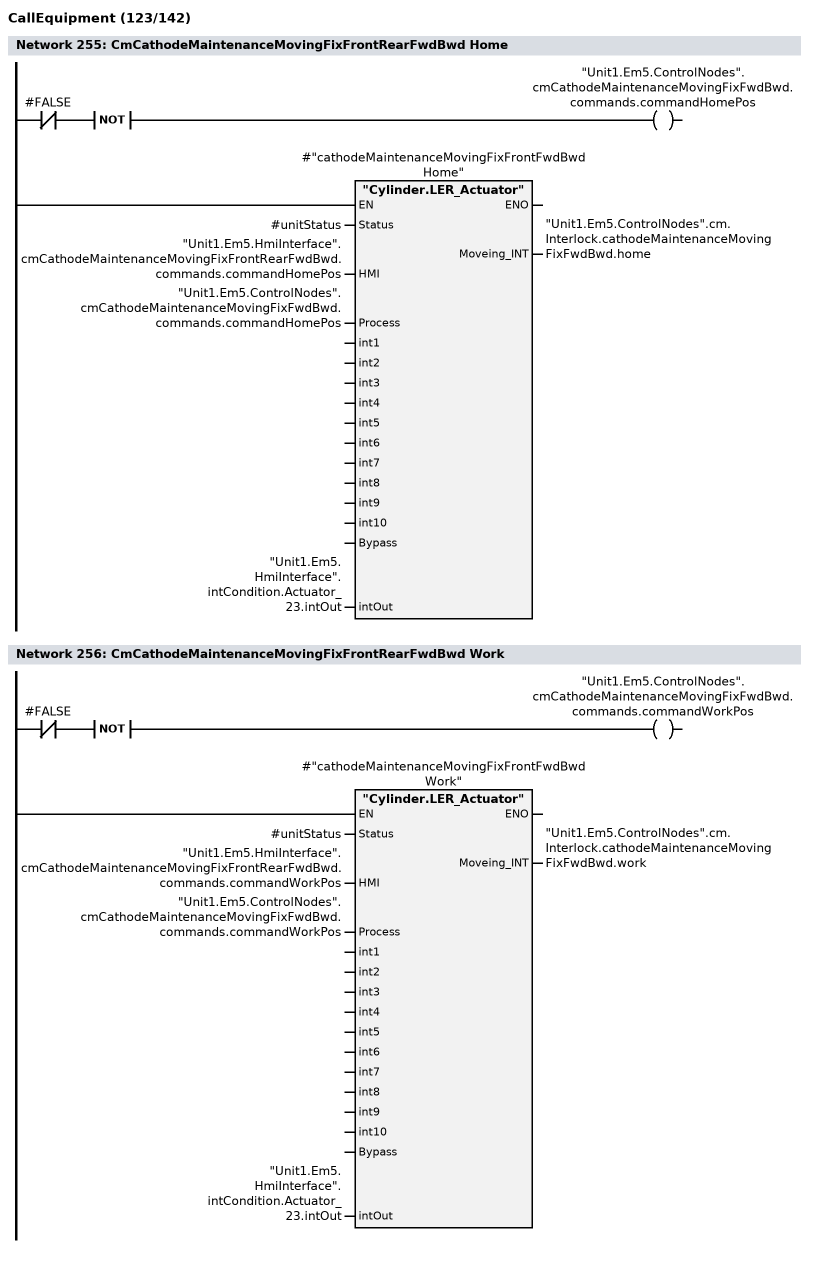
   RUNG wire#powerrail
      I_Contact( #FALSE )
      Not()
      Coil( "Unit1.Em5.ControlNodes".cmCathodeMaintenanceMovingFixFwdBwd.commands.commandHomePos )
   END_RUNG
   RUNG wire#powerrail
      #"cathodeMaintenanceMovingFixFrontFwdBwd Home"(Status := #unitStatus, HMI := "Unit1.Em5.HmiInterface".cmCathodeMaintenanceMovingFixFrontRearFwdBwd.commands.commandHomePos, Process := "Unit1.Em5.ControlNodes".cmCathodeMaintenanceMovingFixFwdBwd.commands.commandHomePos, int1 :=, int2 :=, int3 :=, int4 :=, int5 :=, int6 :=, int7 :=, int8 :=, int9 :=, int10 :=, Bypass :=, intOut := "Unit1.Em5.HmiInterface".intCondition.Actuator_23.intOut, Moveing_INT => "Unit1.Em5.ControlNodes".cm.Interlock.cathodeMaintenanceMovingFixFwdBwd.home)
   END_RUNG
   // the same network as SCL:
   "Unit1.Em5.ControlNodes".cmCathodeMaintenanceMovingFixFwdBwd.commands.commandHomePos := NOT (NOT #FALSE);
   #"cathodeMaintenanceMovingFixFrontFwdBwd Home"(Status := #unitStatus,   // "Cylinder.LER_Actuator"
                           HMI := "Unit1.Em5.HmiInterface".cmCathodeMaintenanceMovingFixFrontRearFwdBwd.commands.commandHomePos,
                           Process := "Unit1.Em5.ControlNodes".cmCathodeMaintenanceMovingFixFwdBwd.commands.commandHomePos,
                           intOut := "Unit1.Em5.HmiInterface".intCondition.Actuator_23.intOut,
                           Moveing_INT => "Unit1.Em5.ControlNodes".cm.Interlock.cathodeMaintenanceMovingFixFwdBwd.home);
END_REGION

REGION Network 256: CmCathodeMaintenanceMovingFixFrontRearFwdBwd Work
   RUNG wire#powerrail
      I_Contact( #FALSE )
      Not()
      Coil( "Unit1.Em5.ControlNodes".cmCathodeMaintenanceMovingFixFwdBwd.commands.commandWorkPos )
   END_RUNG
   RUNG wire#powerrail
      #"cathodeMaintenanceMovingFixFrontFwdBwd Work"(Status := #unitStatus, HMI := "Unit1.Em5.HmiInterface".cmCathodeMaintenanceMovingFixFrontRearFwdBwd.commands.commandWorkPos, Process := "Unit1.Em5.ControlNodes".cmCathodeMaintenanceMovingFixFwdBwd.commands.commandWorkPos, int1 :=, int2 :=, int3 :=, int4 :=, int5 :=, int6 :=, int7 :=, int8 :=, int9 :=, int10 :=, Bypass :=, intOut := "Unit1.Em5.HmiInterface".intCondition.Actuator_23.intOut, Moveing_INT => "Unit1.Em5.ControlNodes".cm.Interlock.cathodeMaintenanceMovingFixFwdBwd.work)
   END_RUNG
   // the same network as SCL:
   "Unit1.Em5.ControlNodes".cmCathodeMaintenanceMovingFixFwdBwd.commands.commandWorkPos := NOT (NOT #FALSE);
   #"cathodeMaintenanceMovingFixFrontFwdBwd Work"(Status := #unitStatus,   // "Cylinder.LER_Actuator"
                           HMI := "Unit1.Em5.HmiInterface".cmCathodeMaintenanceMovingFixFrontRearFwdBwd.commands.commandWorkPos,
                           Process := "Unit1.Em5.ControlNodes".cmCathodeMaintenanceMovingFixFwdBwd.commands.commandWorkPos,
                           intOut := "Unit1.Em5.HmiInterface".intCondition.Actuator_23.intOut,
                           Moveing_INT => "Unit1.Em5.ControlNodes".cm.Interlock.cathodeMaintenanceMovingFixFwdBwd.work);
END_REGION

REGION Network 257: Call instCmCathodeMaintenanceMovingFixFrontRearFwdBwd
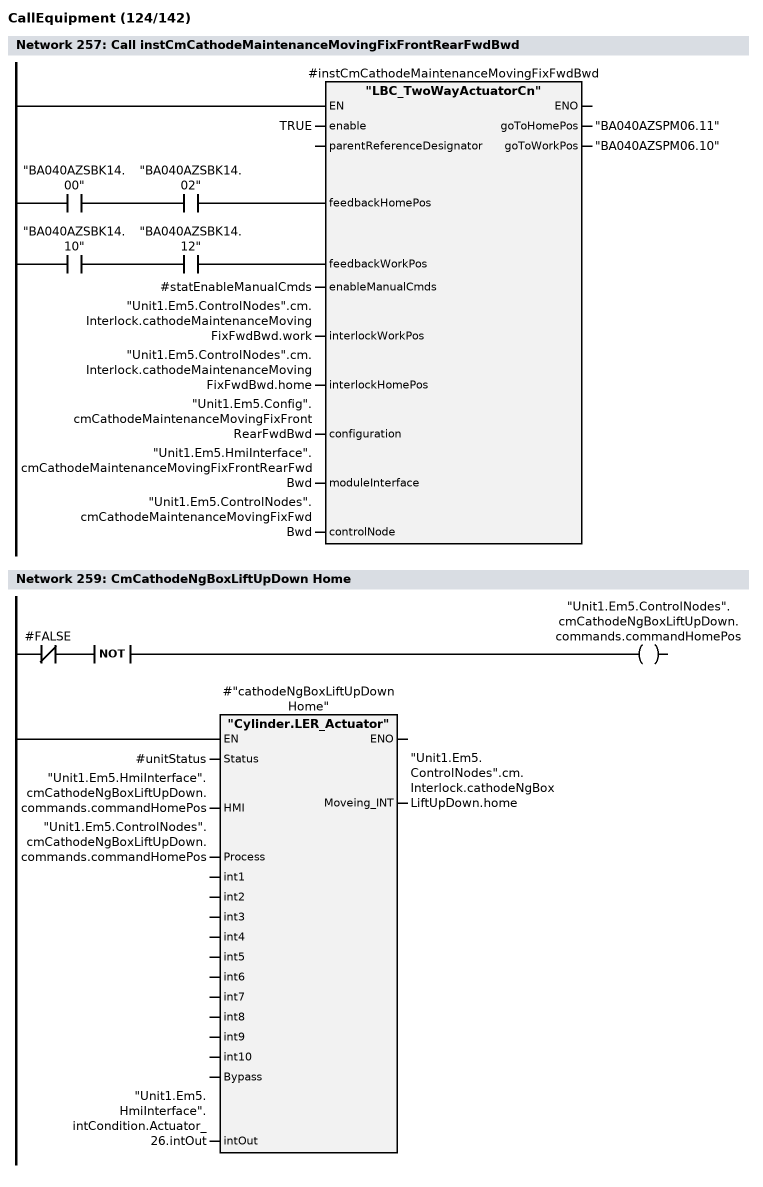
   RUNG wire#powerrail
      #instCmCathodeMaintenanceMovingFixFwdBwd(feedbackHomePos := wire#w1, feedbackWorkPos := wire#w2, enable := TRUE, parentReferenceDesignator :=, enableManualCmds := #statEnableManualCmds, interlockWorkPos := "Unit1.Em5.ControlNodes".cm.Interlock.cathodeMaintenanceMovingFixFwdBwd.work, interlockHomePos := "Unit1.Em5.ControlNodes".cm.Interlock.cathodeMaintenanceMovingFixFwdBwd.home, configuration := "Unit1.Em5.Config".cmCathodeMaintenanceMovingFixFrontRearFwdBwd, moduleInterface := "Unit1.Em5.HmiInterface".cmCathodeMaintenanceMovingFixFrontRearFwdBwd, controlNode := "Unit1.Em5.ControlNodes".cmCathodeMaintenanceMovingFixFwdBwd, goToHomePos => "BA040AZSPM06.11", goToWorkPos => "BA040AZSPM06.10")
   END_RUNG
   RUNG wire#powerrail
      Contact( "BA040AZSBK14.00" )
      Contact( "BA040AZSBK14.02" )
   END_RUNG wire#w1
   RUNG wire#powerrail
      Contact( "BA040AZSBK14.10" )
      Contact( "BA040AZSBK14.12" )
   END_RUNG wire#w2
   // the same network as SCL:
   #instCmCathodeMaintenanceMovingFixFwdBwd(enable := TRUE,   // "LBC_TwoWayActuatorCn"
                           feedbackHomePos := "BA040AZSBK14.00" AND "BA040AZSBK14.02",
                           feedbackWorkPos := "BA040AZSBK14.10" AND "BA040AZSBK14.12",
                           enableManualCmds := #statEnableManualCmds,
                           interlockWorkPos := "Unit1.Em5.ControlNodes".cm.Interlock.cathodeMaintenanceMovingFixFwdBwd.work,
                           interlockHomePos := "Unit1.Em5.ControlNodes".cm.Interlock.cathodeMaintenanceMovingFixFwdBwd.home,
                           configuration := "Unit1.Em5.Config".cmCathodeMaintenanceMovingFixFrontRearFwdBwd,
                           moduleInterface := "Unit1.Em5.HmiInterface".cmCathodeMaintenanceMovingFixFrontRearFwdBwd,
                           controlNode := "Unit1.Em5.ControlNodes".cmCathodeMaintenanceMovingFixFwdBwd,
                           goToHomePos => "BA040AZSPM06.11",
                           goToWorkPos => "BA040AZSPM06.10");
END_REGION

REGION Network 259: CmCathodeNgBoxLiftUpDown Home
   RUNG wire#powerrail
      I_Contact( #FALSE )
      Not()
      Coil( "Unit1.Em5.ControlNodes".cmCathodeNgBoxLiftUpDown.commands.commandHomePos )
   END_RUNG
   RUNG wire#powerrail
      #"cathodeNgBoxLiftUpDown Home"(Status := #unitStatus, HMI := "Unit1.Em5.HmiInterface".cmCathodeNgBoxLiftUpDown.commands.commandHomePos, Process := "Unit1.Em5.ControlNodes".cmCathodeNgBoxLiftUpDown.commands.commandHomePos, int1 :=, int2 :=, int3 :=, int4 :=, int5 :=, int6 :=, int7 :=, int8 :=, int9 :=, int10 :=, Bypass :=, intOut := "Unit1.Em5.HmiInterface".intCondition.Actuator_26.intOut, Moveing_INT => "Unit1.Em5.ControlNodes".cm.Interlock.cathodeNgBoxLiftUpDown.home)
   END_RUNG
   // the same network as SCL:
   "Unit1.Em5.ControlNodes".cmCathodeNgBoxLiftUpDown.commands.commandHomePos := NOT (NOT #FALSE);
   #"cathodeNgBoxLiftUpDown Home"(Status := #unitStatus,   // "Cylinder.LER_Actuator"
                           HMI := "Unit1.Em5.HmiInterface".cmCathodeNgBoxLiftUpDown.commands.commandHomePos,
                           Process := "Unit1.Em5.ControlNodes".cmCathodeNgBoxLiftUpDown.commands.commandHomePos,
                           intOut := "Unit1.Em5.HmiInterface".intCondition.Actuator_26.intOut,
                           Moveing_INT => "Unit1.Em5.ControlNodes".cm.Interlock.cathodeNgBoxLiftUpDown.home);
END_REGION

REGION Network 260: CmCathodeNgBoxLiftUpDown Work
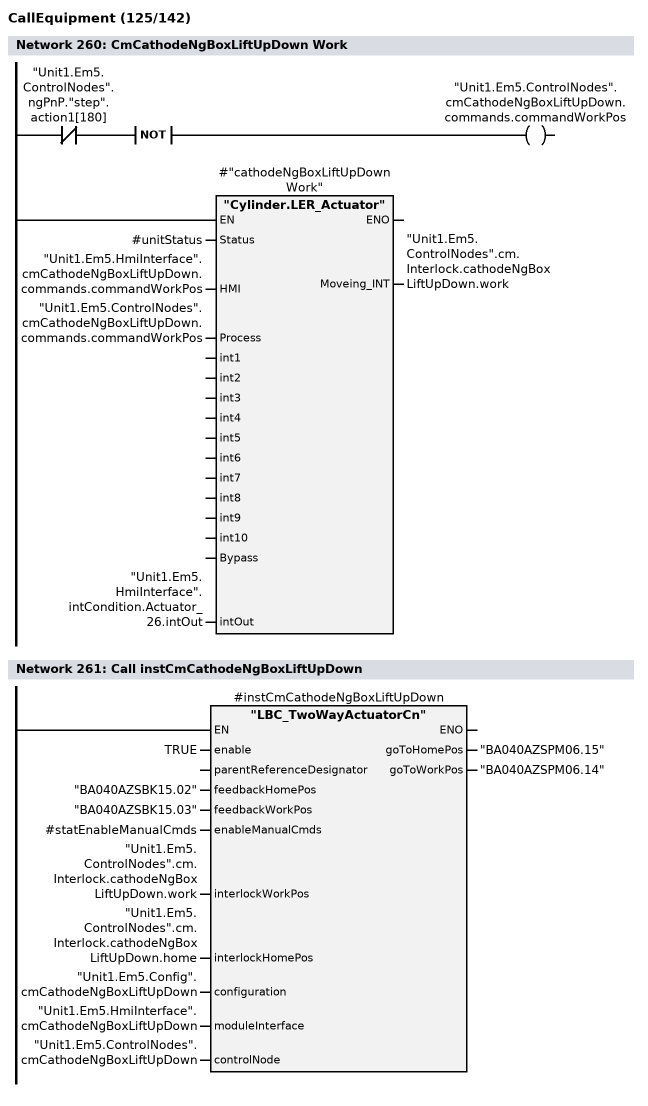
   RUNG wire#powerrail
      I_Contact( "Unit1.Em5.ControlNodes".ngPnP."step".action1[180] )
      Not()
      Coil( "Unit1.Em5.ControlNodes".cmCathodeNgBoxLiftUpDown.commands.commandWorkPos )
   END_RUNG
   RUNG wire#powerrail
      #"cathodeNgBoxLiftUpDown Work"(Status := #unitStatus, HMI := "Unit1.Em5.HmiInterface".cmCathodeNgBoxLiftUpDown.commands.commandWorkPos, Process := "Unit1.Em5.ControlNodes".cmCathodeNgBoxLiftUpDown.commands.commandWorkPos, int1 :=, int2 :=, int3 :=, int4 :=, int5 :=, int6 :=, int7 :=, int8 :=, int9 :=, int10 :=, Bypass :=, intOut := "Unit1.Em5.HmiInterface".intCondition.Actuator_26.intOut, Moveing_INT => "Unit1.Em5.ControlNodes".cm.Interlock.cathodeNgBoxLiftUpDown.work)
   END_RUNG
   // the same network as SCL:
   "Unit1.Em5.ControlNodes".cmCathodeNgBoxLiftUpDown.commands.commandWorkPos := NOT (NOT "Unit1.Em5.ControlNodes".ngPnP."step".action1[180]);
   #"cathodeNgBoxLiftUpDown Work"(Status := #unitStatus,   // "Cylinder.LER_Actuator"
                           HMI := "Unit1.Em5.HmiInterface".cmCathodeNgBoxLiftUpDown.commands.commandWorkPos,
                           Process := "Unit1.Em5.ControlNodes".cmCathodeNgBoxLiftUpDown.commands.commandWorkPos,
                           intOut := "Unit1.Em5.HmiInterface".intCondition.Actuator_26.intOut,
                           Moveing_INT => "Unit1.Em5.ControlNodes".cm.Interlock.cathodeNgBoxLiftUpDown.work);
END_REGION

REGION Network 261: Call instCmCathodeNgBoxLiftUpDown
   RUNG wire#powerrail
      #instCmCathodeNgBoxLiftUpDown(enable := TRUE, parentReferenceDesignator :=, feedbackHomePos := "BA040AZSBK15.02", feedbackWorkPos := "BA040AZSBK15.03", enableManualCmds := #statEnableManualCmds, interlockWorkPos := "Unit1.Em5.ControlNodes".cm.Interlock.cathodeNgBoxLiftUpDown.work, interlockHomePos := "Unit1.Em5.ControlNodes".cm.Interlock.cathodeNgBoxLiftUpDown.home, configuration := "Unit1.Em5.Config".cmCathodeNgBoxLiftUpDown, moduleInterface := "Unit1.Em5.HmiInterface".cmCathodeNgBoxLiftUpDown, controlNode := "Unit1.Em5.ControlNodes".cmCathodeNgBoxLiftUpDown, goToHomePos => "BA040AZSPM06.15", goToWorkPos => "BA040AZSPM06.14")
   END_RUNG
   // the same network as SCL:
   #instCmCathodeNgBoxLiftUpDown(enable := TRUE,   // "LBC_TwoWayActuatorCn"
                           feedbackHomePos := "BA040AZSBK15.02",
                           feedbackWorkPos := "BA040AZSBK15.03",
                           enableManualCmds := #statEnableManualCmds,
                           interlockWorkPos := "Unit1.Em5.ControlNodes".cm.Interlock.cathodeNgBoxLiftUpDown.work,
                           interlockHomePos := "Unit1.Em5.ControlNodes".cm.Interlock.cathodeNgBoxLiftUpDown.home,
                           configuration := "Unit1.Em5.Config".cmCathodeNgBoxLiftUpDown,
                           moduleInterface := "Unit1.Em5.HmiInterface".cmCathodeNgBoxLiftUpDown,
                           controlNode := "Unit1.Em5.ControlNodes".cmCathodeNgBoxLiftUpDown,
                           goToHomePos => "BA040AZSPM06.15",
                           goToWorkPos => "BA040AZSPM06.14");
END_REGION

REGION Network 263: CmCathodeNgBoxLockUpDown Home
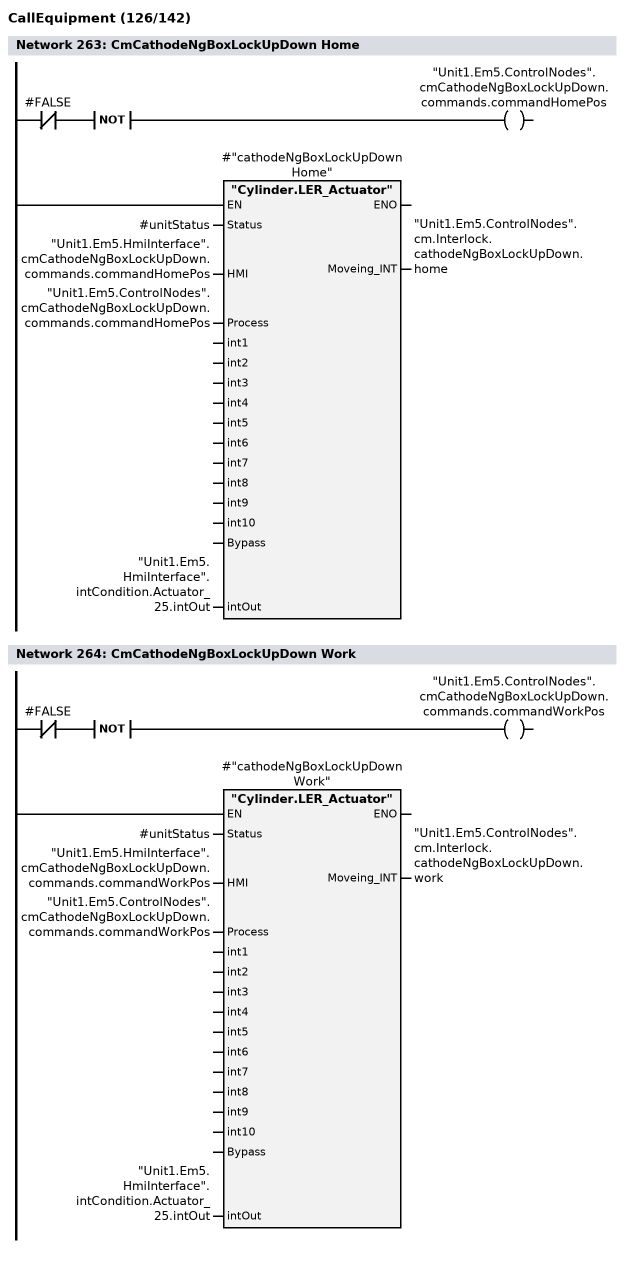
   RUNG wire#powerrail
      I_Contact( #FALSE )
      Not()
      Coil( "Unit1.Em5.ControlNodes".cmCathodeNgBoxLockUpDown.commands.commandHomePos )
   END_RUNG
   RUNG wire#powerrail
      #"cathodeNgBoxLockUpDown Home"(Status := #unitStatus, HMI := "Unit1.Em5.HmiInterface".cmCathodeNgBoxLockUpDown.commands.commandHomePos, Process := "Unit1.Em5.ControlNodes".cmCathodeNgBoxLockUpDown.commands.commandHomePos, int1 :=, int2 :=, int3 :=, int4 :=, int5 :=, int6 :=, int7 :=, int8 :=, int9 :=, int10 :=, Bypass :=, intOut := "Unit1.Em5.HmiInterface".intCondition.Actuator_25.intOut, Moveing_INT => "Unit1.Em5.ControlNodes".cm.Interlock.cathodeNgBoxLockUpDown.home)
   END_RUNG
   // the same network as SCL:
   "Unit1.Em5.ControlNodes".cmCathodeNgBoxLockUpDown.commands.commandHomePos := NOT (NOT #FALSE);
   #"cathodeNgBoxLockUpDown Home"(Status := #unitStatus,   // "Cylinder.LER_Actuator"
                           HMI := "Unit1.Em5.HmiInterface".cmCathodeNgBoxLockUpDown.commands.commandHomePos,
                           Process := "Unit1.Em5.ControlNodes".cmCathodeNgBoxLockUpDown.commands.commandHomePos,
                           intOut := "Unit1.Em5.HmiInterface".intCondition.Actuator_25.intOut,
                           Moveing_INT => "Unit1.Em5.ControlNodes".cm.Interlock.cathodeNgBoxLockUpDown.home);
END_REGION

REGION Network 264: CmCathodeNgBoxLockUpDown Work
   RUNG wire#powerrail
      I_Contact( #FALSE )
      Not()
      Coil( "Unit1.Em5.ControlNodes".cmCathodeNgBoxLockUpDown.commands.commandWorkPos )
   END_RUNG
   RUNG wire#powerrail
      #"cathodeNgBoxLockUpDown Work"(Status := #unitStatus, HMI := "Unit1.Em5.HmiInterface".cmCathodeNgBoxLockUpDown.commands.commandWorkPos, Process := "Unit1.Em5.ControlNodes".cmCathodeNgBoxLockUpDown.commands.commandWorkPos, int1 :=, int2 :=, int3 :=, int4 :=, int5 :=, int6 :=, int7 :=, int8 :=, int9 :=, int10 :=, Bypass :=, intOut := "Unit1.Em5.HmiInterface".intCondition.Actuator_25.intOut, Moveing_INT => "Unit1.Em5.ControlNodes".cm.Interlock.cathodeNgBoxLockUpDown.work)
   END_RUNG
   // the same network as SCL:
   "Unit1.Em5.ControlNodes".cmCathodeNgBoxLockUpDown.commands.commandWorkPos := NOT (NOT #FALSE);
   #"cathodeNgBoxLockUpDown Work"(Status := #unitStatus,   // "Cylinder.LER_Actuator"
                           HMI := "Unit1.Em5.HmiInterface".cmCathodeNgBoxLockUpDown.commands.commandWorkPos,
                           Process := "Unit1.Em5.ControlNodes".cmCathodeNgBoxLockUpDown.commands.commandWorkPos,
                           intOut := "Unit1.Em5.HmiInterface".intCondition.Actuator_25.intOut,
                           Moveing_INT => "Unit1.Em5.ControlNodes".cm.Interlock.cathodeNgBoxLockUpDown.work);
END_REGION

REGION Network 265: Call instCmCathodeNgBoxLockUpDown
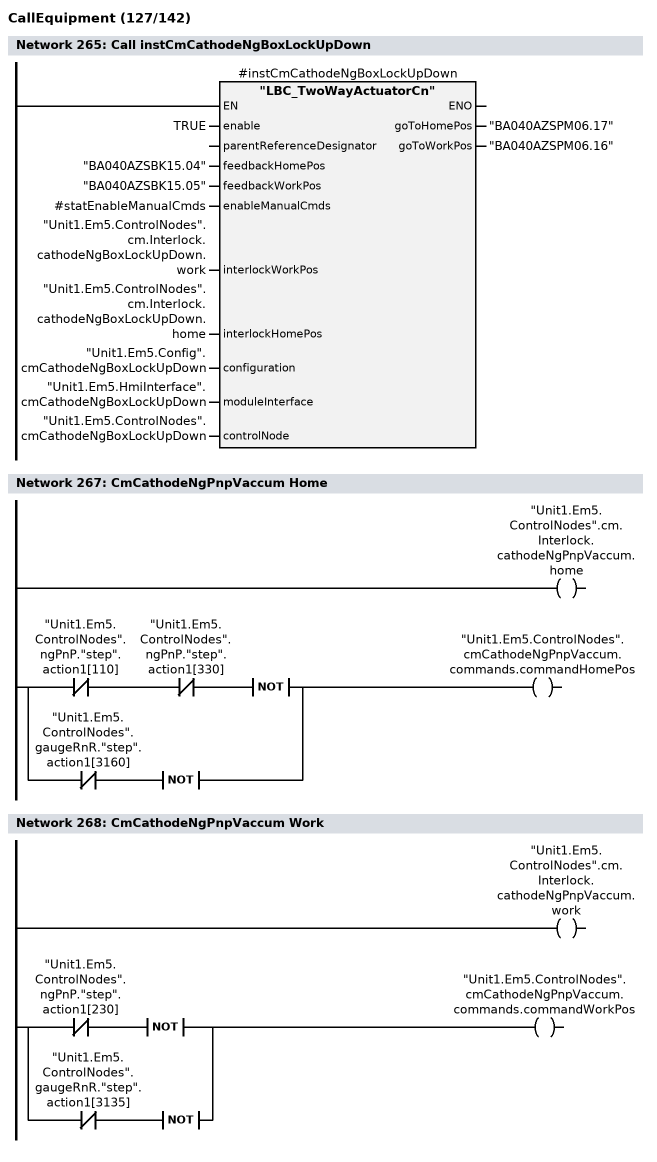
   RUNG wire#powerrail
      #instCmCathodeNgBoxLockUpDown(enable := TRUE, parentReferenceDesignator :=, feedbackHomePos := "BA040AZSBK15.04", feedbackWorkPos := "BA040AZSBK15.05", enableManualCmds := #statEnableManualCmds, interlockWorkPos := "Unit1.Em5.ControlNodes".cm.Interlock.cathodeNgBoxLockUpDown.work, interlockHomePos := "Unit1.Em5.ControlNodes".cm.Interlock.cathodeNgBoxLockUpDown.home, configuration := "Unit1.Em5.Config".cmCathodeNgBoxLockUpDown, moduleInterface := "Unit1.Em5.HmiInterface".cmCathodeNgBoxLockUpDown, controlNode := "Unit1.Em5.ControlNodes".cmCathodeNgBoxLockUpDown, goToHomePos => "BA040AZSPM06.17", goToWorkPos => "BA040AZSPM06.16")
   END_RUNG
   // the same network as SCL:
   #instCmCathodeNgBoxLockUpDown(enable := TRUE,   // "LBC_TwoWayActuatorCn"
                           feedbackHomePos := "BA040AZSBK15.04",
                           feedbackWorkPos := "BA040AZSBK15.05",
                           enableManualCmds := #statEnableManualCmds,
                           interlockWorkPos := "Unit1.Em5.ControlNodes".cm.Interlock.cathodeNgBoxLockUpDown.work,
                           interlockHomePos := "Unit1.Em5.ControlNodes".cm.Interlock.cathodeNgBoxLockUpDown.home,
                           configuration := "Unit1.Em5.Config".cmCathodeNgBoxLockUpDown,
                           moduleInterface := "Unit1.Em5.HmiInterface".cmCathodeNgBoxLockUpDown,
                           controlNode := "Unit1.Em5.ControlNodes".cmCathodeNgBoxLockUpDown,
                           goToHomePos => "BA040AZSPM06.17",
                           goToWorkPos => "BA040AZSPM06.16");
END_REGION

REGION Network 267: CmCathodeNgPnpVaccum Home
   RUNG wire#powerrail
      Coil( "Unit1.Em5.ControlNodes".cm.Interlock.cathodeNgPnpVaccum.home )
   END_RUNG
   RUNG wire#powerrail
      I_Contact( "Unit1.Em5.ControlNodes".ngPnP."step".action1[110] )
      I_Contact( "Unit1.Em5.ControlNodes".ngPnP."step".action1[330] )
      Not()
      wire#w1
      Coil( "Unit1.Em5.ControlNodes".cmCathodeNgPnpVaccum.commands.commandHomePos )
   END_RUNG
   RUNG wire#powerrail
      I_Contact( "Unit1.Em5.ControlNodes".gaugeRnR."step".action1[3160] )
      Not()
   END_RUNG wire#w1
   // the same network as SCL:
   "Unit1.Em5.ControlNodes".cm.Interlock.cathodeNgPnpVaccum.home := TRUE;
   "Unit1.Em5.ControlNodes".cmCathodeNgPnpVaccum.commands.commandHomePos := NOT (NOT "Unit1.Em5.ControlNodes".ngPnP."step".action1[110] AND NOT "Unit1.Em5.ControlNodes".ngPnP."step".action1[330]) OR NOT (NOT "Unit1.Em5.ControlNodes".gaugeRnR."step".action1[3160]);
END_REGION

REGION Network 268: CmCathodeNgPnpVaccum Work
   RUNG wire#powerrail
      Coil( "Unit1.Em5.ControlNodes".cm.Interlock.cathodeNgPnpVaccum.work )
   END_RUNG
   RUNG wire#powerrail
      I_Contact( "Unit1.Em5.ControlNodes".ngPnP."step".action1[230] )
      Not()
      wire#w1
      Coil( "Unit1.Em5.ControlNodes".cmCathodeNgPnpVaccum.commands.commandWorkPos )
   END_RUNG
   RUNG wire#powerrail
      I_Contact( "Unit1.Em5.ControlNodes".gaugeRnR."step".action1[3135] )
      Not()
   END_RUNG wire#w1
   // the same network as SCL:
   "Unit1.Em5.ControlNodes".cm.Interlock.cathodeNgPnpVaccum.work := TRUE;
   "Unit1.Em5.ControlNodes".cmCathodeNgPnpVaccum.commands.commandWorkPos := NOT (NOT "Unit1.Em5.ControlNodes".ngPnP."step".action1[230]) OR NOT (NOT "Unit1.Em5.ControlNodes".gaugeRnR."step".action1[3135]);
END_REGION

REGION Network 269: Call instCmCathodeNgPnpVaccum
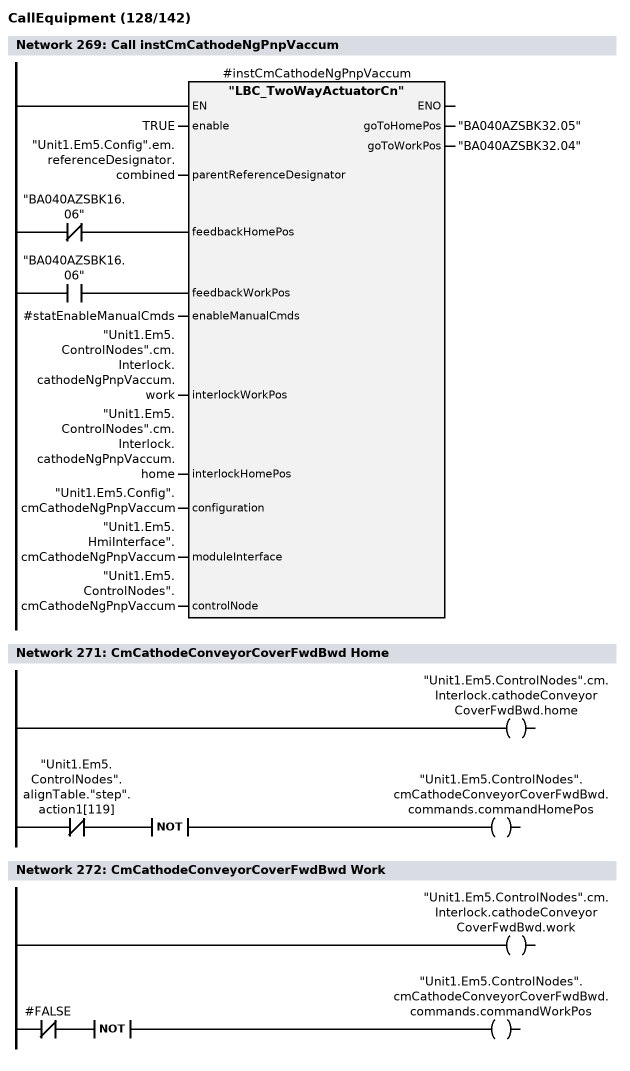
   RUNG wire#powerrail
      #instCmCathodeNgPnpVaccum(feedbackHomePos := wire#w1, feedbackWorkPos := wire#w2, enable := TRUE, parentReferenceDesignator := "Unit1.Em5.Config".em.referenceDesignator.combined, enableManualCmds := #statEnableManualCmds, interlockWorkPos := "Unit1.Em5.ControlNodes".cm.Interlock.cathodeNgPnpVaccum.work, interlockHomePos := "Unit1.Em5.ControlNodes".cm.Interlock.cathodeNgPnpVaccum.home, configuration := "Unit1.Em5.Config".cmCathodeNgPnpVaccum, moduleInterface := "Unit1.Em5.HmiInterface".cmCathodeNgPnpVaccum, controlNode := "Unit1.Em5.ControlNodes".cmCathodeNgPnpVaccum, goToHomePos => "BA040AZSBK32.05", goToWorkPos => "BA040AZSBK32.04")
   END_RUNG
   RUNG wire#powerrail
      I_Contact( "BA040AZSBK16.06" )
   END_RUNG wire#w1
   RUNG wire#powerrail
      Contact( "BA040AZSBK16.06" )
   END_RUNG wire#w2
   // the same network as SCL:
   #instCmCathodeNgPnpVaccum(enable := TRUE,   // "LBC_TwoWayActuatorCn"
                           parentReferenceDesignator := "Unit1.Em5.Config".em.referenceDesignator.combined,
                           feedbackHomePos := NOT "BA040AZSBK16.06",
                           feedbackWorkPos := "BA040AZSBK16.06",
                           enableManualCmds := #statEnableManualCmds,
                           interlockWorkPos := "Unit1.Em5.ControlNodes".cm.Interlock.cathodeNgPnpVaccum.work,
                           interlockHomePos := "Unit1.Em5.ControlNodes".cm.Interlock.cathodeNgPnpVaccum.home,
                           configuration := "Unit1.Em5.Config".cmCathodeNgPnpVaccum,
                           moduleInterface := "Unit1.Em5.HmiInterface".cmCathodeNgPnpVaccum,
                           controlNode := "Unit1.Em5.ControlNodes".cmCathodeNgPnpVaccum,
                           goToHomePos => "BA040AZSBK32.05",
                           goToWorkPos => "BA040AZSBK32.04");
END_REGION

REGION Network 271: CmCathodeConveyorCoverFwdBwd Home
   RUNG wire#powerrail
      Coil( "Unit1.Em5.ControlNodes".cm.Interlock.cathodeConveyorCoverFwdBwd.home )
   END_RUNG
   RUNG wire#powerrail
      I_Contact( "Unit1.Em5.ControlNodes".alignTable."step".action1[119] )
      Not()
      Coil( "Unit1.Em5.ControlNodes".cmCathodeConveyorCoverFwdBwd.commands.commandHomePos )
   END_RUNG
   // the same network as SCL:
   "Unit1.Em5.ControlNodes".cm.Interlock.cathodeConveyorCoverFwdBwd.home := TRUE;
   "Unit1.Em5.ControlNodes".cmCathodeConveyorCoverFwdBwd.commands.commandHomePos := NOT (NOT "Unit1.Em5.ControlNodes".alignTable."step".action1[119]);
END_REGION

REGION Network 272: CmCathodeConveyorCoverFwdBwd Work
   RUNG wire#powerrail
      Coil( "Unit1.Em5.ControlNodes".cm.Interlock.cathodeConveyorCoverFwdBwd.work )
   END_RUNG
   RUNG wire#powerrail
      I_Contact( #FALSE )
      Not()
      Coil( "Unit1.Em5.ControlNodes".cmCathodeConveyorCoverFwdBwd.commands.commandWorkPos )
   END_RUNG
   // the same network as SCL:
   "Unit1.Em5.ControlNodes".cm.Interlock.cathodeConveyorCoverFwdBwd.work := TRUE;
   "Unit1.Em5.ControlNodes".cmCathodeConveyorCoverFwdBwd.commands.commandWorkPos := NOT (NOT #FALSE);
END_REGION

REGION Network 273: Call instCmCathodeConveyorCoverFwdBwd
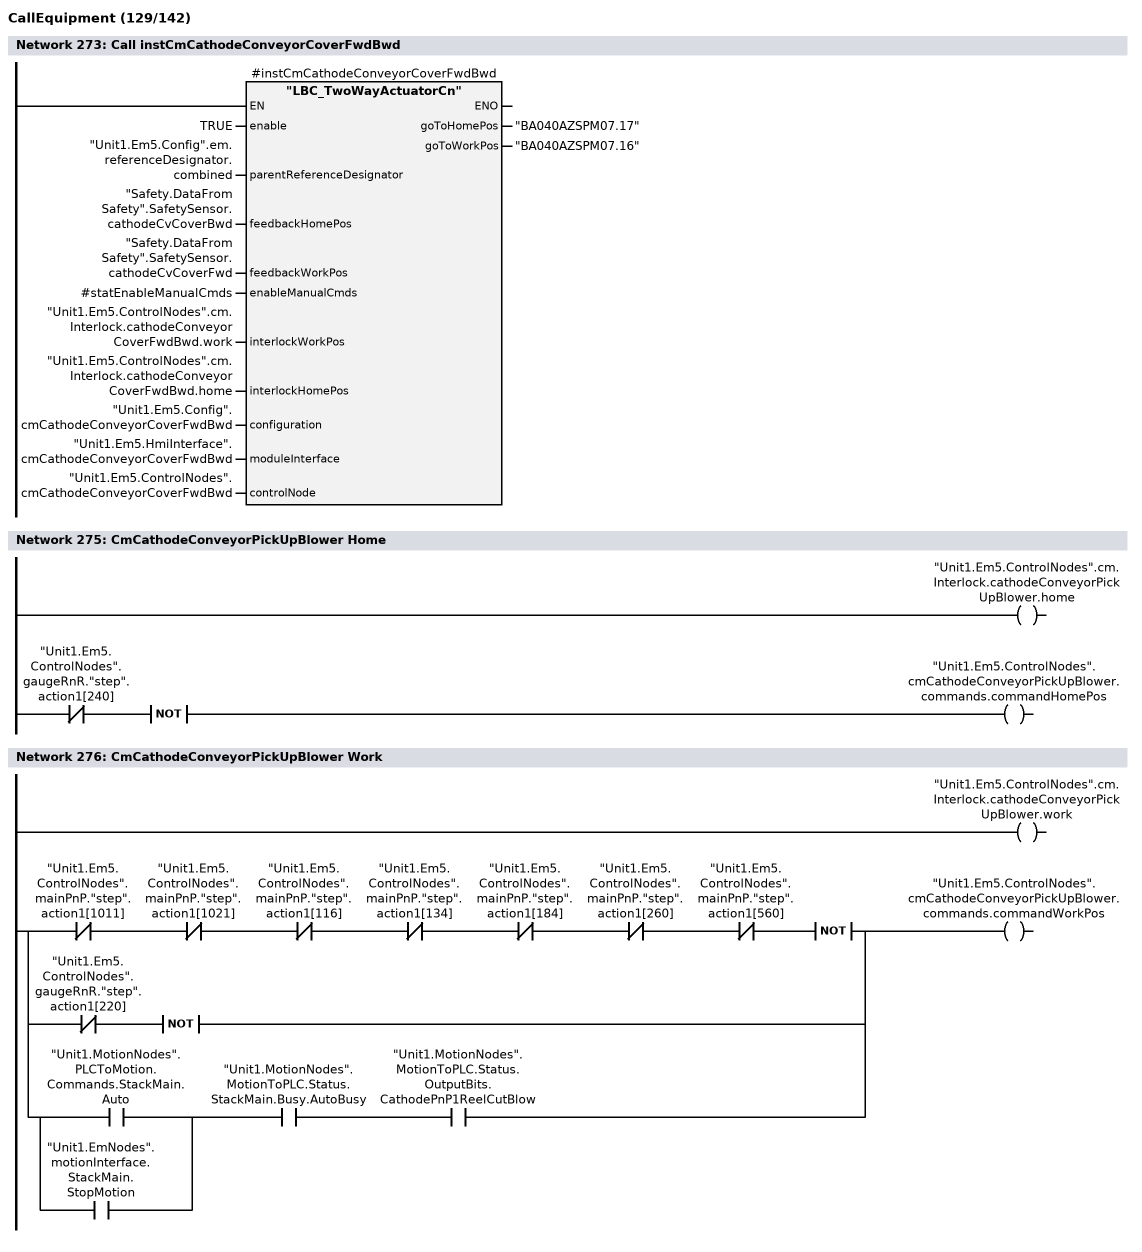
   RUNG wire#powerrail
      #instCmCathodeConveyorCoverFwdBwd(enable := TRUE, parentReferenceDesignator := "Unit1.Em5.Config".em.referenceDesignator.combined, feedbackHomePos := "Safety.DataFromSafety".SafetySensor.cathodeCvCoverBwd, feedbackWorkPos := "Safety.DataFromSafety".SafetySensor.cathodeCvCoverFwd, enableManualCmds := #statEnableManualCmds, interlockWorkPos := "Unit1.Em5.ControlNodes".cm.Interlock.cathodeConveyorCoverFwdBwd.work, interlockHomePos := "Unit1.Em5.ControlNodes".cm.Interlock.cathodeConveyorCoverFwdBwd.home, configuration := "Unit1.Em5.Config".cmCathodeConveyorCoverFwdBwd, moduleInterface := "Unit1.Em5.HmiInterface".cmCathodeConveyorCoverFwdBwd, controlNode := "Unit1.Em5.ControlNodes".cmCathodeConveyorCoverFwdBwd, goToHomePos => "BA040AZSPM07.17", goToWorkPos => "BA040AZSPM07.16")
   END_RUNG
   // the same network as SCL:
   #instCmCathodeConveyorCoverFwdBwd(enable := TRUE,   // "LBC_TwoWayActuatorCn"
                           parentReferenceDesignator := "Unit1.Em5.Config".em.referenceDesignator.combined,
                           feedbackHomePos := "Safety.DataFromSafety".SafetySensor.cathodeCvCoverBwd,
                           feedbackWorkPos := "Safety.DataFromSafety".SafetySensor.cathodeCvCoverFwd,
                           enableManualCmds := #statEnableManualCmds,
                           interlockWorkPos := "Unit1.Em5.ControlNodes".cm.Interlock.cathodeConveyorCoverFwdBwd.work,
                           interlockHomePos := "Unit1.Em5.ControlNodes".cm.Interlock.cathodeConveyorCoverFwdBwd.home,
                           configuration := "Unit1.Em5.Config".cmCathodeConveyorCoverFwdBwd,
                           moduleInterface := "Unit1.Em5.HmiInterface".cmCathodeConveyorCoverFwdBwd,
                           controlNode := "Unit1.Em5.ControlNodes".cmCathodeConveyorCoverFwdBwd,
                           goToHomePos => "BA040AZSPM07.17",
                           goToWorkPos => "BA040AZSPM07.16");
END_REGION

REGION Network 275: CmCathodeConveyorPickUpBlower Home
   RUNG wire#powerrail
      Coil( "Unit1.Em5.ControlNodes".cm.Interlock.cathodeConveyorPickUpBlower.home )
   END_RUNG
   RUNG wire#powerrail
      I_Contact( "Unit1.Em5.ControlNodes".gaugeRnR."step".action1[240] )
      Not()
      Coil( "Unit1.Em5.ControlNodes".cmCathodeConveyorPickUpBlower.commands.commandHomePos )
   END_RUNG
   // the same network as SCL:
   "Unit1.Em5.ControlNodes".cm.Interlock.cathodeConveyorPickUpBlower.home := TRUE;
   "Unit1.Em5.ControlNodes".cmCathodeConveyorPickUpBlower.commands.commandHomePos := NOT (NOT "Unit1.Em5.ControlNodes".gaugeRnR."step".action1[240]);
END_REGION

REGION Network 276: CmCathodeConveyorPickUpBlower Work
   RUNG wire#powerrail
      Coil( "Unit1.Em5.ControlNodes".cm.Interlock.cathodeConveyorPickUpBlower.work )
   END_RUNG
   RUNG wire#powerrail
      I_Contact( "Unit1.Em5.ControlNodes".mainPnP."step".action1[1011] )
      I_Contact( "Unit1.Em5.ControlNodes".mainPnP."step".action1[1021] )
      I_Contact( "Unit1.Em5.ControlNodes".mainPnP."step".action1[116] )
      I_Contact( "Unit1.Em5.ControlNodes".mainPnP."step".action1[134] )
      I_Contact( "Unit1.Em5.ControlNodes".mainPnP."step".action1[184] )
      I_Contact( "Unit1.Em5.ControlNodes".mainPnP."step".action1[260] )
      I_Contact( "Unit1.Em5.ControlNodes".mainPnP."step".action1[560] )
      Not()
      wire#w1
      Coil( "Unit1.Em5.ControlNodes".cmCathodeConveyorPickUpBlower.commands.commandWorkPos )
   END_RUNG
   RUNG wire#powerrail
      I_Contact( "Unit1.Em5.ControlNodes".gaugeRnR."step".action1[220] )
      Not()
   END_RUNG wire#w1
   RUNG wire#powerrail
      Contact( "Unit1.MotionNodes".PLCToMotion.Commands.StackMain.Auto )
      wire#w2
      Contact( "Unit1.MotionNodes".MotionToPLC.Status.StackMain.Busy.AutoBusy )
      Contact( "Unit1.MotionNodes".MotionToPLC.Status.OutputBits.CathodePnP1ReelCutBlow )
   END_RUNG wire#w1
   RUNG wire#powerrail
      Contact( "Unit1.EmNodes".motionInterface.StackMain.StopMotion )
   END_RUNG wire#w2
   // the same network as SCL:
   "Unit1.Em5.ControlNodes".cm.Interlock.cathodeConveyorPickUpBlower.work := TRUE;
   "Unit1.Em5.ControlNodes".cmCathodeConveyorPickUpBlower.commands.commandWorkPos := NOT (NOT "Unit1.Em5.ControlNodes".mainPnP."step".action1[1011] AND NOT "Unit1.Em5.ControlNodes".mainPnP."step".action1[1021] AND NOT "Unit1.Em5.ControlNodes".mainPnP."step".action1[116] AND NOT "Unit1.Em5.ControlNodes".mainPnP."step".action1[134] AND NOT "Unit1.Em5.ControlNodes".mainPnP."step".action1[184] AND NOT "Unit1.Em5.ControlNodes".mainPnP."step".action1[260] AND NOT "Unit1.Em5.ControlNodes".mainPnP."step".action1[560]) OR NOT (NOT "Unit1.Em5.ControlNodes".gaugeRnR."step".action1[220]) OR (("Unit1.MotionNodes".PLCToMotion.Commands.StackMain.Auto OR "Unit1.EmNodes".motionInterface.StackMain.StopMotion) AND "Unit1.MotionNodes".MotionToPLC.Status.StackMain.Busy.AutoBusy AND "Unit1.MotionNodes".MotionToPLC.Status.OutputBits.CathodePnP1ReelCutBlow);
END_REGION

REGION Network 277: Call instCmCathodeConveyorPickUpBlower
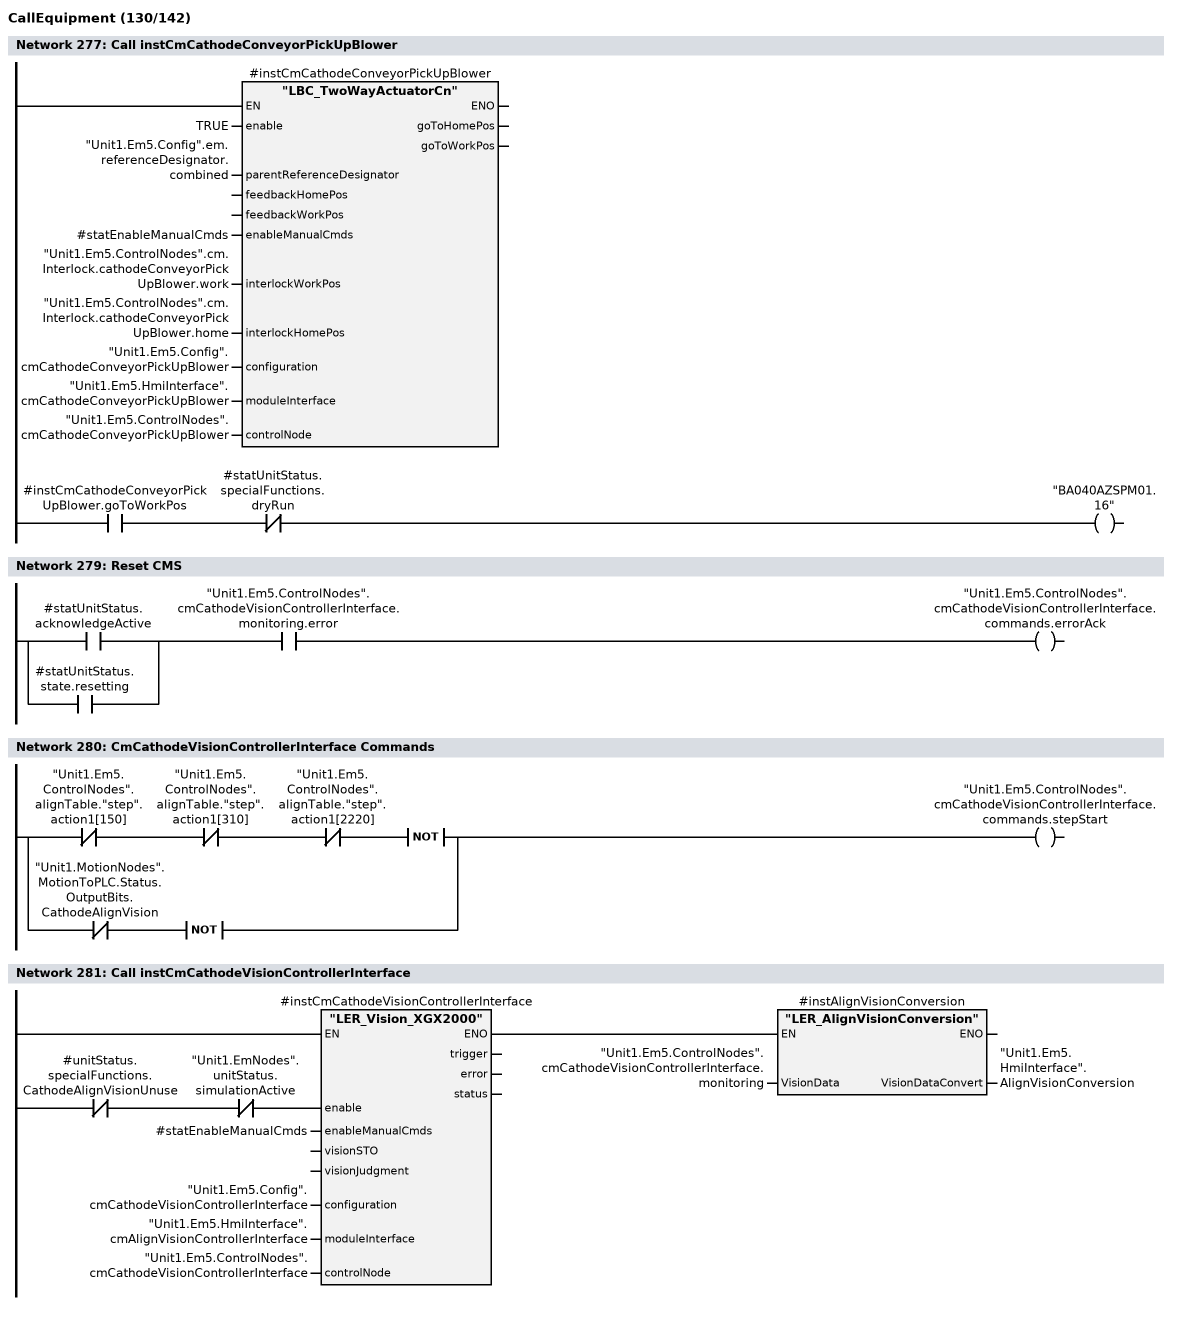
   RUNG wire#powerrail
      #instCmCathodeConveyorPickUpBlower(enable := TRUE, parentReferenceDesignator := "Unit1.Em5.Config".em.referenceDesignator.combined, feedbackHomePos :=, feedbackWorkPos :=, enableManualCmds := #statEnableManualCmds, interlockWorkPos := "Unit1.Em5.ControlNodes".cm.Interlock.cathodeConveyorPickUpBlower.work, interlockHomePos := "Unit1.Em5.ControlNodes".cm.Interlock.cathodeConveyorPickUpBlower.home, configuration := "Unit1.Em5.Config".cmCathodeConveyorPickUpBlower, moduleInterface := "Unit1.Em5.HmiInterface".cmCathodeConveyorPickUpBlower, controlNode := "Unit1.Em5.ControlNodes".cmCathodeConveyorPickUpBlower, goToHomePos =>, goToWorkPos =>)
   END_RUNG
   RUNG wire#powerrail
      Contact( #instCmCathodeConveyorPickUpBlower.goToWorkPos )
      I_Contact( #statUnitStatus.specialFunctions.dryRun )
      Coil( "BA040AZSPM01.16" )
   END_RUNG
   // the same network as SCL:
   #instCmCathodeConveyorPickUpBlower(enable := TRUE,   // "LBC_TwoWayActuatorCn"
                           parentReferenceDesignator := "Unit1.Em5.Config".em.referenceDesignator.combined,
                           enableManualCmds := #statEnableManualCmds,
                           interlockWorkPos := "Unit1.Em5.ControlNodes".cm.Interlock.cathodeConveyorPickUpBlower.work,
                           interlockHomePos := "Unit1.Em5.ControlNodes".cm.Interlock.cathodeConveyorPickUpBlower.home,
                           configuration := "Unit1.Em5.Config".cmCathodeConveyorPickUpBlower,
                           moduleInterface := "Unit1.Em5.HmiInterface".cmCathodeConveyorPickUpBlower,
                           controlNode := "Unit1.Em5.ControlNodes".cmCathodeConveyorPickUpBlower);
   "BA040AZSPM01.16" := #instCmCathodeConveyorPickUpBlower.goToWorkPos AND NOT #statUnitStatus.specialFunctions.dryRun;
END_REGION

REGION Network 278: ******************** Control Modules (Accessories) ********************
END_REGION

REGION Network 279: Reset CMS
   RUNG wire#powerrail
      Contact( #statUnitStatus.acknowledgeActive )
      wire#w1
      Contact( "Unit1.Em5.ControlNodes".cmCathodeVisionControllerInterface.monitoring.error )
      Coil( "Unit1.Em5.ControlNodes".cmCathodeVisionControllerInterface.commands.errorAck )
   END_RUNG
   RUNG wire#powerrail
      Contact( #statUnitStatus.state.resetting )
   END_RUNG wire#w1
   // the same network as SCL:
   "Unit1.Em5.ControlNodes".cmCathodeVisionControllerInterface.commands.errorAck := (#statUnitStatus.acknowledgeActive OR #statUnitStatus.state.resetting) AND "Unit1.Em5.ControlNodes".cmCathodeVisionControllerInterface.monitoring.error;
END_REGION

REGION Network 280: CmCathodeVisionControllerInterface Commands
   RUNG wire#powerrail
      I_Contact( "Unit1.Em5.ControlNodes".alignTable."step".action1[150] )
      I_Contact( "Unit1.Em5.ControlNodes".alignTable."step".action1[310] )
      I_Contact( "Unit1.Em5.ControlNodes".alignTable."step".action1[2220] )
      Not()
      wire#w1
      Coil( "Unit1.Em5.ControlNodes".cmCathodeVisionControllerInterface.commands.stepStart )
   END_RUNG
   RUNG wire#powerrail
      I_Contact( "Unit1.MotionNodes".MotionToPLC.Status.OutputBits.CathodeAlignVision )
      Not()
   END_RUNG wire#w1
   // the same network as SCL:
   "Unit1.Em5.ControlNodes".cmCathodeVisionControllerInterface.commands.stepStart := NOT (NOT "Unit1.Em5.ControlNodes".alignTable."step".action1[150] AND NOT "Unit1.Em5.ControlNodes".alignTable."step".action1[310] AND NOT "Unit1.Em5.ControlNodes".alignTable."step".action1[2220]) OR NOT (NOT "Unit1.MotionNodes".MotionToPLC.Status.OutputBits.CathodeAlignVision);
END_REGION

REGION Network 281: Call instCmCathodeVisionControllerInterface
   RUNG wire#powerrail
      #instCmCathodeVisionControllerInterface(enable := wire#w1, enableManualCmds := #statEnableManualCmds, visionSTO :=, visionJudgment :=, configuration := "Unit1.Em5.Config".cmCathodeVisionControllerInterface, moduleInterface := "Unit1.Em5.HmiInterface".cmAlignVisionControllerInterface, controlNode := "Unit1.Em5.ControlNodes".cmCathodeVisionControllerInterface, trigger =>, error =>, status =>)
      #instAlignVisionConversion(VisionData := "Unit1.Em5.ControlNodes".cmCathodeVisionControllerInterface.monitoring, VisionDataConvert => "Unit1.Em5.HmiInterface".AlignVisionConversion)
   END_RUNG
   RUNG wire#powerrail
      I_Contact( #unitStatus.specialFunctions.CathodeAlignVisionUnuse )
      I_Contact( "Unit1.EmNodes".unitStatus.simulationActive )
   END_RUNG wire#w1
   // the same network as SCL:
   #instCmCathodeVisionControllerInterface(enable := NOT #unitStatus.specialFunctions.CathodeAlignVisionUnuse AND NOT "Unit1.EmNodes".unitStatus.simulationActive,   // "LER_Vision_XGX2000"
                           enableManualCmds := #statEnableManualCmds,
                           configuration := "Unit1.Em5.Config".cmCathodeVisionControllerInterface,
                           moduleInterface := "Unit1.Em5.HmiInterface".cmAlignVisionControllerInterface,
                           controlNode := "Unit1.Em5.ControlNodes".cmCathodeVisionControllerInterface,
                           ENO => #_w1);
   IF #_w1 THEN
       #instAlignVisionConversion(VisionData := "Unit1.Em5.ControlNodes".cmCathodeVisionControllerInterface.monitoring,   // "LER_AlignVisionConversion"
                               VisionDataConvert => "Unit1.Em5.HmiInterface".AlignVisionConversion);
   END_IF;
END_REGION

REGION Network 282: *************** Feedback to Unit ***************************
END_REGION

REGION Network 283: Determine StateComplete (SC) in Mode Production
   // Conditions for the Equipment Modules "stateComplete" feedback to the unit. This feedback is given when the task in for the respective state is complete.
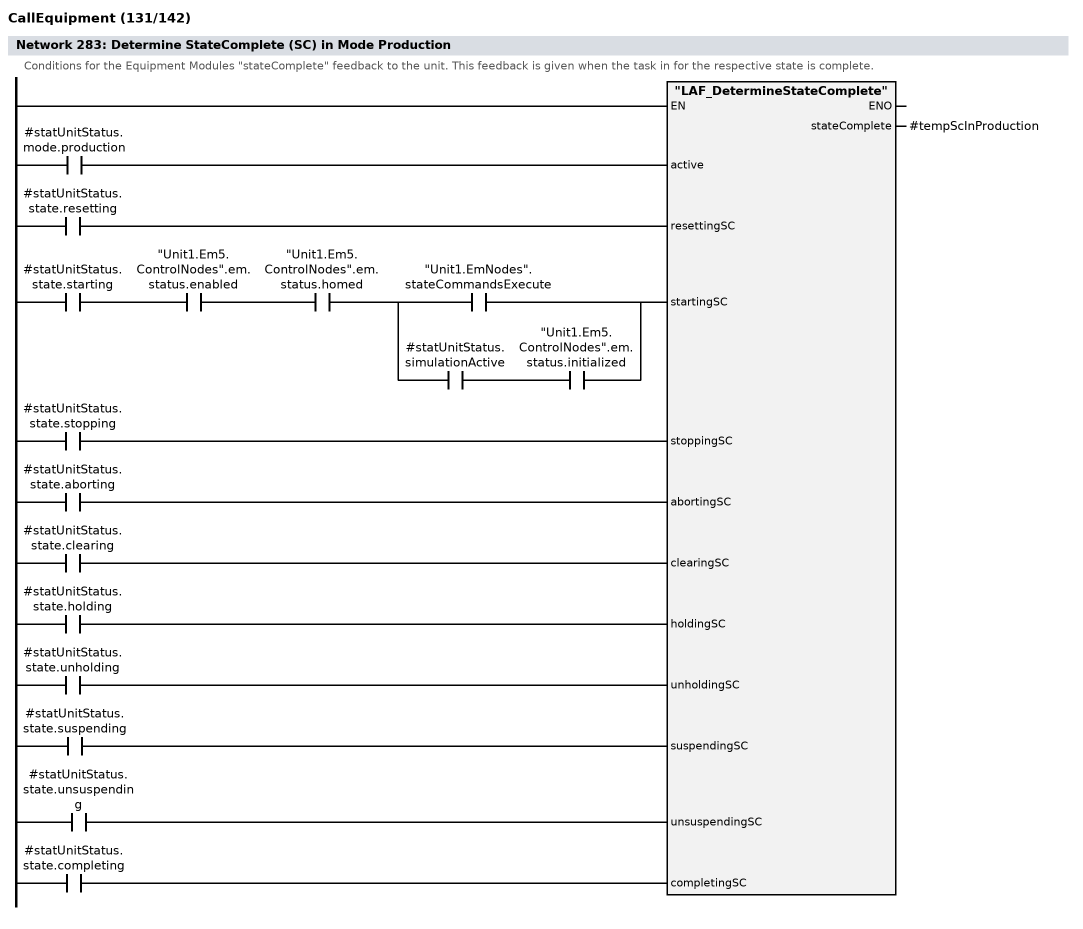
   RUNG wire#powerrail
      "LAF_DetermineStateComplete"(active := wire#w1, resettingSC := wire#w2, startingSC := wire#w4, stoppingSC := wire#w5, abortingSC := wire#w6, clearingSC := wire#w7, holdingSC := wire#w8, unholdingSC := wire#w9, suspendingSC := wire#w10, unsuspendingSC := wire#w11, completingSC := wire#w12, stateComplete => #tempScInProduction)
   END_RUNG
   RUNG wire#powerrail
      Contact( #statUnitStatus.mode.production )
   END_RUNG wire#w1
   RUNG wire#powerrail
      Contact( #statUnitStatus.state.resetting )
   END_RUNG wire#w2
   RUNG wire#powerrail
      Contact( #statUnitStatus.state.starting )
      Contact( "Unit1.Em5.ControlNodes".em.status.enabled )
      Contact( "Unit1.Em5.ControlNodes".em.status.homed )
      wire#w3
      Contact( "Unit1.EmNodes".stateCommandsExecute )
   END_RUNG wire#w4
   RUNG wire#w3
      Contact( #statUnitStatus.simulationActive )
      Contact( "Unit1.Em5.ControlNodes".em.status.initialized )
   END_RUNG wire#w4
   RUNG wire#powerrail
      Contact( #statUnitStatus.state.stopping )
   END_RUNG wire#w5
   RUNG wire#powerrail
      Contact( #statUnitStatus.state.aborting )
   END_RUNG wire#w6
   RUNG wire#powerrail
      Contact( #statUnitStatus.state.clearing )
   END_RUNG wire#w7
   RUNG wire#powerrail
      Contact( #statUnitStatus.state.holding )
   END_RUNG wire#w8
   RUNG wire#powerrail
      Contact( #statUnitStatus.state.unholding )
   END_RUNG wire#w9
   RUNG wire#powerrail
      Contact( #statUnitStatus.state.suspending )
   END_RUNG wire#w10
   RUNG wire#powerrail
      Contact( #statUnitStatus.state.unsuspending )
   END_RUNG wire#w11
   RUNG wire#powerrail
      Contact( #statUnitStatus.state.completing )
   END_RUNG wire#w12
   // the same network as SCL:
   "LAF_DetermineStateComplete"(active := #statUnitStatus.mode.production,
                           resettingSC := #statUnitStatus.state.resetting,
                           startingSC := #statUnitStatus.state.starting AND "Unit1.Em5.ControlNodes".em.status.enabled AND "Unit1.Em5.ControlNodes".em.status.homed AND ("Unit1.EmNodes".stateCommandsExecute OR (#statUnitStatus.simulationActive AND "Unit1.Em5.ControlNodes".em.status.initialized)),
                           stoppingSC := #statUnitStatus.state.stopping,
                           abortingSC := #statUnitStatus.state.aborting,
                           clearingSC := #statUnitStatus.state.clearing,
                           holdingSC := #statUnitStatus.state.holding,
                           unholdingSC := #statUnitStatus.state.unholding,
                           suspendingSC := #statUnitStatus.state.suspending,
                           unsuspendingSC := #statUnitStatus.state.unsuspending,
                           completingSC := #statUnitStatus.state.completing,
                           stateComplete => #tempScInProduction);
END_REGION

REGION Network 284: Determine StateComplete (SC) in Mode Maintenance/Manual
   // Conditions for the Equipment Modules "stateComplete" feedback to the unit. This feedback is given when the task in for the respective state is complete.
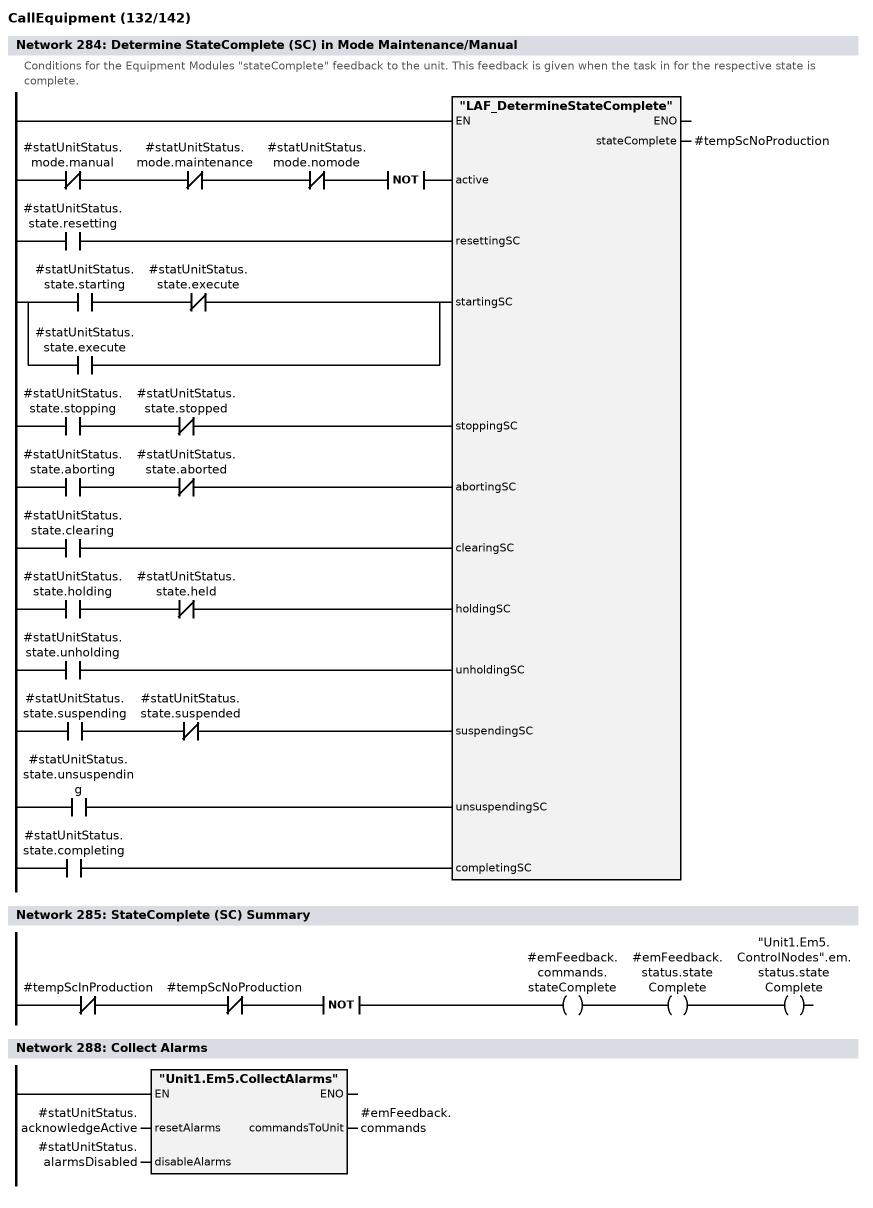
   RUNG wire#powerrail
      "LAF_DetermineStateComplete"(active := wire#w1, resettingSC := wire#w2, startingSC := wire#w3, stoppingSC := wire#w4, abortingSC := wire#w5, clearingSC := wire#w6, holdingSC := wire#w7, unholdingSC := wire#w8, suspendingSC := wire#w9, unsuspendingSC := wire#w10, completingSC := wire#w11, stateComplete => #tempScNoProduction)
   END_RUNG
   RUNG wire#powerrail
      I_Contact( #statUnitStatus.mode.manual )
      I_Contact( #statUnitStatus.mode.maintenance )
      I_Contact( #statUnitStatus.mode.nomode )
      Not()
   END_RUNG wire#w1
   RUNG wire#powerrail
      Contact( #statUnitStatus.state.resetting )
   END_RUNG wire#w2
   RUNG wire#powerrail
      Contact( #statUnitStatus.state.starting )
      I_Contact( #statUnitStatus.state.execute )
   END_RUNG wire#w3
   RUNG wire#powerrail
      Contact( #statUnitStatus.state.execute )
   END_RUNG wire#w3
   RUNG wire#powerrail
      Contact( #statUnitStatus.state.stopping )
      I_Contact( #statUnitStatus.state.stopped )
   END_RUNG wire#w4
   RUNG wire#powerrail
      Contact( #statUnitStatus.state.aborting )
      I_Contact( #statUnitStatus.state.aborted )
   END_RUNG wire#w5
   RUNG wire#powerrail
      Contact( #statUnitStatus.state.clearing )
   END_RUNG wire#w6
   RUNG wire#powerrail
      Contact( #statUnitStatus.state.holding )
      I_Contact( #statUnitStatus.state.held )
   END_RUNG wire#w7
   RUNG wire#powerrail
      Contact( #statUnitStatus.state.unholding )
   END_RUNG wire#w8
   RUNG wire#powerrail
      Contact( #statUnitStatus.state.suspending )
      I_Contact( #statUnitStatus.state.suspended )
   END_RUNG wire#w9
   RUNG wire#powerrail
      Contact( #statUnitStatus.state.unsuspending )
   END_RUNG wire#w10
   RUNG wire#powerrail
      Contact( #statUnitStatus.state.completing )
   END_RUNG wire#w11
   // the same network as SCL:
   "LAF_DetermineStateComplete"(active := NOT (NOT #statUnitStatus.mode.manual AND NOT #statUnitStatus.mode.maintenance AND NOT #statUnitStatus.mode.nomode),
                           resettingSC := #statUnitStatus.state.resetting,
                           startingSC := (#statUnitStatus.state.starting AND NOT #statUnitStatus.state.execute) OR #statUnitStatus.state.execute,
                           stoppingSC := #statUnitStatus.state.stopping AND NOT #statUnitStatus.state.stopped,
                           abortingSC := #statUnitStatus.state.aborting AND NOT #statUnitStatus.state.aborted,
                           clearingSC := #statUnitStatus.state.clearing,
                           holdingSC := #statUnitStatus.state.holding AND NOT #statUnitStatus.state.held,
                           unholdingSC := #statUnitStatus.state.unholding,
                           suspendingSC := #statUnitStatus.state.suspending AND NOT #statUnitStatus.state.suspended,
                           unsuspendingSC := #statUnitStatus.state.unsuspending,
                           completingSC := #statUnitStatus.state.completing,
                           stateComplete => #tempScNoProduction);
END_REGION

REGION Network 285: StateComplete (SC) Summary
   RUNG wire#powerrail
      I_Contact( #tempScInProduction )
      I_Contact( #tempScNoProduction )
      Not()
      Coil( #emFeedback.commands.stateComplete )
      Coil( #emFeedback.status.stateComplete )
      Coil( "Unit1.Em5.ControlNodes".em.status.stateComplete )
   END_RUNG
   // the same network as SCL:
   #emFeedback.commands.stateComplete := NOT (NOT #tempScInProduction AND NOT #tempScNoProduction);
   #emFeedback.status.stateComplete := #emFeedback.commands.stateComplete;
   "Unit1.Em5.ControlNodes".em.status.stateComplete := #emFeedback.commands.stateComplete;
END_REGION

REGION Network 287: *************** Alarms **********************************
END_REGION

REGION Network 288: Collect Alarms
   RUNG wire#powerrail
      "Unit1.Em5.CollectAlarms"(resetAlarms := #statUnitStatus.acknowledgeActive, disableAlarms := #statUnitStatus.alarmsDisabled, commandsToUnit => #emFeedback.commands)
   END_RUNG
   // the same network as SCL:
   "Unit1.Em5.CollectAlarms"(resetAlarms := #statUnitStatus.acknowledgeActive,
                           disableAlarms := #statUnitStatus.alarmsDisabled,
                           commandsToUnit => #emFeedback.commands);
END_REGION

REGION Network 289: Manage Alarms
   // Derive commands from the ProDiag supervision. The ProDiag supervisions contain categories which define the reaction of these supervisions (e.g. abort, stop, hold). These are handed over as commands to the unit level.
   // Alternatively, if no ProDiag should be used, you can use the LAF_ManageBitAlarms to realize bit alarm handling. This block can be found in LAF in folder 70_AlarmHandling.
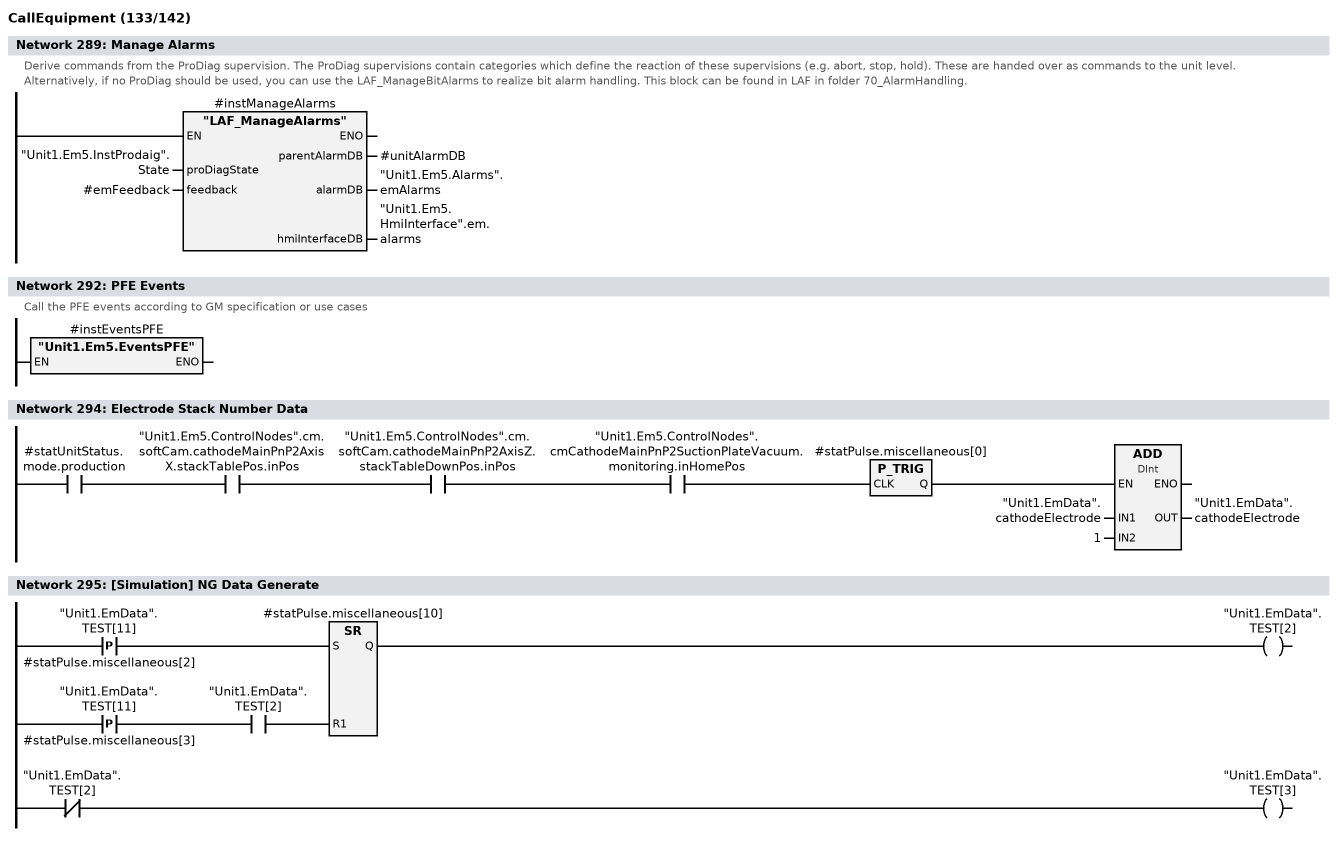
   RUNG wire#powerrail
      #instManageAlarms(proDiagState := "Unit1.Em5.InstProdaig".State, feedback := #emFeedback, parentAlarmDB => #unitAlarmDB, alarmDB => "Unit1.Em5.Alarms".emAlarms, hmiInterfaceDB => "Unit1.Em5.HmiInterface".em.alarms)
   END_RUNG
   // the same network as SCL:
   #instManageAlarms(proDiagState := "Unit1.Em5.InstProdaig".State,   // "LAF_ManageAlarms"
                     feedback := #emFeedback,
                     parentAlarmDB => #unitAlarmDB,
                     alarmDB => "Unit1.Em5.Alarms".emAlarms,
                     hmiInterfaceDB => "Unit1.Em5.HmiInterface".em.alarms);
END_REGION

REGION Network 291: *************** PFE Events**********************************
END_REGION

REGION Network 292: PFE Events
   // Call the PFE events according to GM specification or use cases
   RUNG wire#powerrail
      #instEventsPFE()
   END_RUNG
   // the same network as SCL:
   #instEventsPFE();   // "Unit1.Em5.EventsPFE"
END_REGION

REGION Network 293: ******************** Part Data ********************
END_REGION

REGION Network 294: Electrode Stack Number Data
   RUNG wire#powerrail
      Contact( #statUnitStatus.mode.production )
      Contact( "Unit1.Em5.ControlNodes".cm.softCam.cathodeMainPnP2AxisX.stackTablePos.inPos )
      Contact( "Unit1.Em5.ControlNodes".cm.softCam.cathodeMainPnP2AxisZ.stackTableDownPos.inPos )
      Contact( "Unit1.Em5.ControlNodes".cmCathodeMainPnP2SuctionPlateVacuum.monitoring.inHomePos )
      P_Trig( #statPulse.miscellaneous[0] )
      { S7_Templates := "SrcType := DInt" } Add(in1 := "Unit1.EmData".cathodeElectrode, in2 := 1, out => "Unit1.EmData".cathodeElectrode)
   END_RUNG
   // the same network as SCL:
   #_w1 := #statUnitStatus.mode.production AND "Unit1.Em5.ControlNodes".cm.softCam.cathodeMainPnP2AxisX.stackTablePos.inPos AND "Unit1.Em5.ControlNodes".cm.softCam.cathodeMainPnP2AxisZ.stackTableDownPos.inPos AND "Unit1.Em5.ControlNodes".cmCathodeMainPnP2SuctionPlateVacuum.monitoring.inHomePos;
   #_w2 := #_w1 AND NOT #statPulse.miscellaneous[0];   // rising edge
   #statPulse.miscellaneous[0] := #_w1;
   IF #_w2 THEN "Unit1.EmData".cathodeElectrode := "Unit1.EmData".cathodeElectrode + 1; END_IF;
END_REGION

REGION Network 295: [Simulation] NG Data Generate
   RUNG wire#powerrail
      P_Contact(operand := "Unit1.EmData".TEST[11], bit := #statPulse.miscellaneous[2])
      S_SR(operand := #statPulse.miscellaneous[10], r1 := wire#w1)
      Coil( "Unit1.EmData".TEST[2] )
   END_RUNG
   RUNG wire#powerrail
      P_Contact(operand := "Unit1.EmData".TEST[11], bit := #statPulse.miscellaneous[3])
      Contact( "Unit1.EmData".TEST[2] )
   END_RUNG wire#w1
   RUNG wire#powerrail
      I_Contact( "Unit1.EmData".TEST[2] )
      Coil( "Unit1.EmData".TEST[3] )
   END_RUNG
   // the same network as SCL:
   #_w1 := "Unit1.EmData".TEST[11] AND NOT #statPulse.miscellaneous[2];   // rising edge of "Unit1.EmData".TEST[11]
   #statPulse.miscellaneous[2] := "Unit1.EmData".TEST[11];
   #_w2 := "Unit1.EmData".TEST[11] AND NOT #statPulse.miscellaneous[3];   // rising edge of "Unit1.EmData".TEST[11]
   #statPulse.miscellaneous[3] := "Unit1.EmData".TEST[11];
   IF #_w1 THEN
       #statPulse.miscellaneous[10] := TRUE;   // SR flip-flop
   END_IF;
   IF #_w2 AND "Unit1.EmData".TEST[2] THEN #statPulse.miscellaneous[10] := FALSE; END_IF;
   "Unit1.EmData".TEST[2] := #statPulse.miscellaneous[10];
   "Unit1.EmData".TEST[3] := NOT "Unit1.EmData".TEST[2];
END_REGION

REGION Network 296: Align Vision Data
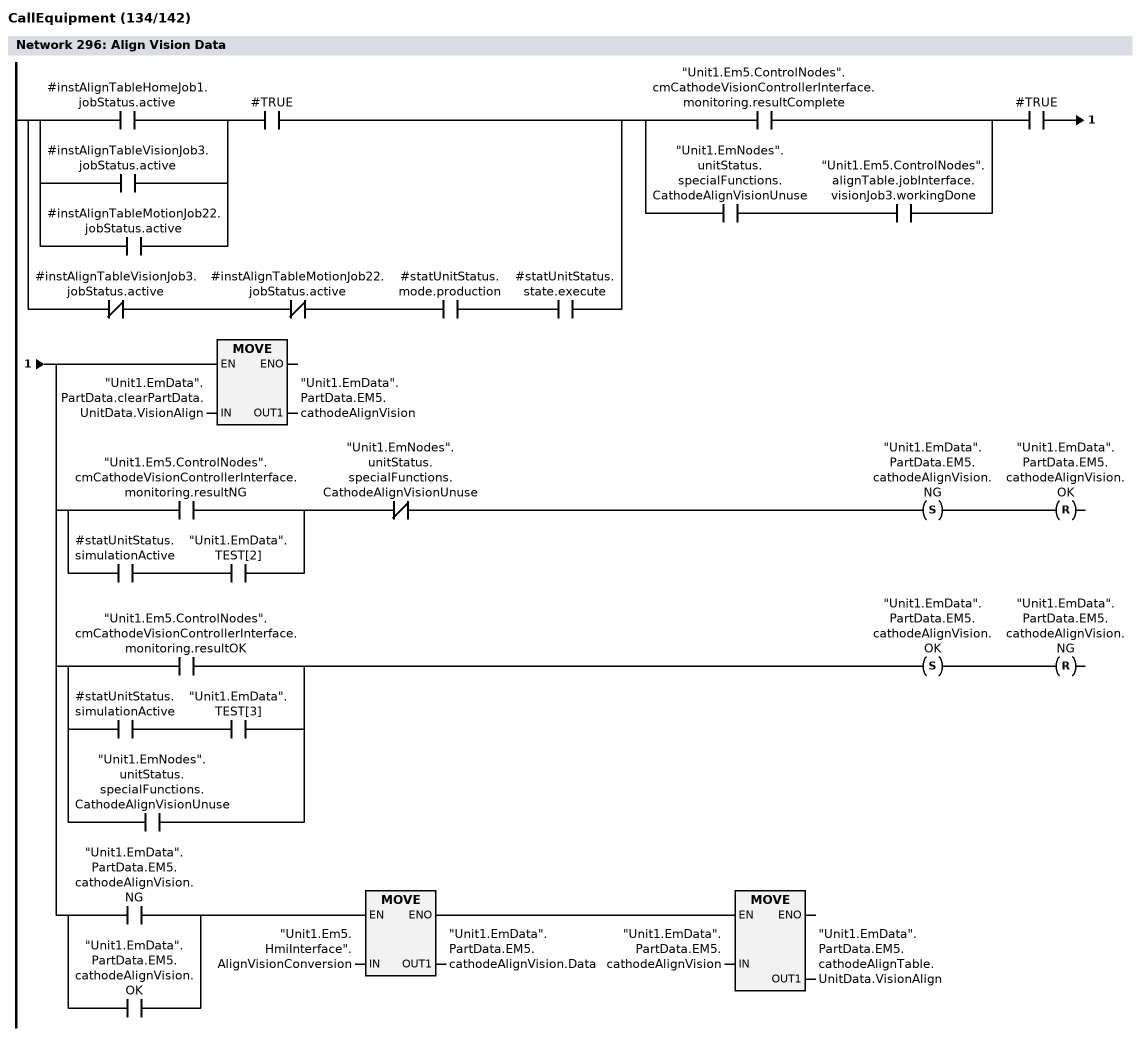
   RUNG wire#powerrail
      Contact( #instAlignTableHomeJob1.jobStatus.active )
      wire#w1
      Contact( #TRUE )
      wire#w2
      Contact( "Unit1.Em5.ControlNodes".cmCathodeVisionControllerInterface.monitoring.resultComplete )
      wire#w3
      Contact( #TRUE )
      wire#w4
      Move(in := "Unit1.EmData".PartData.clearPartData.UnitData.VisionAlign, out1 => "Unit1.EmData".PartData.EM5.cathodeAlignVision)
   END_RUNG
   RUNG wire#powerrail
      Contact( #instAlignTableVisionJob3.jobStatus.active )
   END_RUNG wire#w1
   RUNG wire#powerrail
      Contact( #instAlignTableMotionJob22.jobStatus.active )
   END_RUNG wire#w1
   RUNG wire#powerrail
      I_Contact( #instAlignTableVisionJob3.jobStatus.active )
      I_Contact( #instAlignTableMotionJob22.jobStatus.active )
      Contact( #statUnitStatus.mode.production )
      Contact( #statUnitStatus.state.execute )
   END_RUNG wire#w2
   RUNG wire#w2
      Contact( "Unit1.EmNodes".unitStatus.specialFunctions.CathodeAlignVisionUnuse )
      Contact( "Unit1.Em5.ControlNodes".alignTable.jobInterface.visionJob3.workingDone )
   END_RUNG wire#w3
   RUNG wire#w4
      Contact( "Unit1.Em5.ControlNodes".cmCathodeVisionControllerInterface.monitoring.resultNG )
      wire#w5
      I_Contact( "Unit1.EmNodes".unitStatus.specialFunctions.CathodeAlignVisionUnuse )
      S_Coil( "Unit1.EmData".PartData.EM5.cathodeAlignVision.NG )
      R_Coil( "Unit1.EmData".PartData.EM5.cathodeAlignVision.OK )
   END_RUNG
   RUNG wire#w4
      Contact( #statUnitStatus.simulationActive )
      Contact( "Unit1.EmData".TEST[2] )
   END_RUNG wire#w5
   RUNG wire#w4
      Contact( "Unit1.Em5.ControlNodes".cmCathodeVisionControllerInterface.monitoring.resultOK )
      wire#w6
      S_Coil( "Unit1.EmData".PartData.EM5.cathodeAlignVision.OK )
      R_Coil( "Unit1.EmData".PartData.EM5.cathodeAlignVision.NG )
   END_RUNG
   RUNG wire#w4
      Contact( #statUnitStatus.simulationActive )
      Contact( "Unit1.EmData".TEST[3] )
   END_RUNG wire#w6
   RUNG wire#w4
      Contact( "Unit1.EmNodes".unitStatus.specialFunctions.CathodeAlignVisionUnuse )
   END_RUNG wire#w6
   RUNG wire#w4
      Contact( "Unit1.EmData".PartData.EM5.cathodeAlignVision.NG )
      wire#w7
      Move(in := "Unit1.Em5.HmiInterface".AlignVisionConversion, out1 => "Unit1.EmData".PartData.EM5.cathodeAlignVision.Data)
      Move(in := "Unit1.EmData".PartData.EM5.cathodeAlignVision, out1 => "Unit1.EmData".PartData.EM5.cathodeAlignTable.UnitData.VisionAlign)
   END_RUNG
   RUNG wire#w4
      Contact( "Unit1.EmData".PartData.EM5.cathodeAlignVision.OK )
   END_RUNG wire#w7
   // the same network as SCL:
   #_w1 := (((#instAlignTableHomeJob1.jobStatus.active OR #instAlignTableVisionJob3.jobStatus.active OR #instAlignTableMotionJob22.jobStatus.active) AND #TRUE) OR (NOT #instAlignTableVisionJob3.jobStatus.active AND NOT #instAlignTableMotionJob22.jobStatus.active AND #statUnitStatus.mode.production AND #statUnitStatus.state.execute)) AND ("Unit1.Em5.ControlNodes".cmCathodeVisionControllerInterface.monitoring.resultComplete OR ("Unit1.EmNodes".unitStatus.specialFunctions.CathodeAlignVisionUnuse AND "Unit1.Em5.ControlNodes".alignTable.jobInterface.visionJob3.workingDone)) AND #TRUE;
   IF #_w1 THEN
       "Unit1.EmData".PartData.EM5.cathodeAlignVision := "Unit1.EmData".PartData.clearPartData.UnitData.VisionAlign;
   END_IF;
   IF #_w1 AND ("Unit1.Em5.ControlNodes".cmCathodeVisionControllerInterface.monitoring.resultNG OR (#statUnitStatus.simulationActive AND "Unit1.EmData".TEST[2])) AND NOT "Unit1.EmNodes".unitStatus.specialFunctions.CathodeAlignVisionUnuse THEN
       "Unit1.EmData".PartData.EM5.cathodeAlignVision.NG := TRUE;
       "Unit1.EmData".PartData.EM5.cathodeAlignVision.OK := FALSE;
   END_IF;
   IF #_w1 AND ("Unit1.Em5.ControlNodes".cmCathodeVisionControllerInterface.monitoring.resultOK OR (#statUnitStatus.simulationActive AND "Unit1.EmData".TEST[3]) OR "Unit1.EmNodes".unitStatus.specialFunctions.CathodeAlignVisionUnuse) THEN
       "Unit1.EmData".PartData.EM5.cathodeAlignVision.OK := TRUE;
       "Unit1.EmData".PartData.EM5.cathodeAlignVision.NG := FALSE;
   END_IF;
   IF #_w1 AND ("Unit1.EmData".PartData.EM5.cathodeAlignVision.NG OR "Unit1.EmData".PartData.EM5.cathodeAlignVision.OK) THEN
       "Unit1.EmData".PartData.EM5.cathodeAlignVision.Data := "Unit1.Em5.HmiInterface".AlignVisionConversion;
       "Unit1.EmData".PartData.EM5.cathodeAlignTable.UnitData.VisionAlign := "Unit1.EmData".PartData.EM5.cathodeAlignVision;
   END_IF;
END_REGION

REGION Network 297: ******************** Unit Output ********************
END_REGION

REGION Network 298: Em Nodes Brake Test
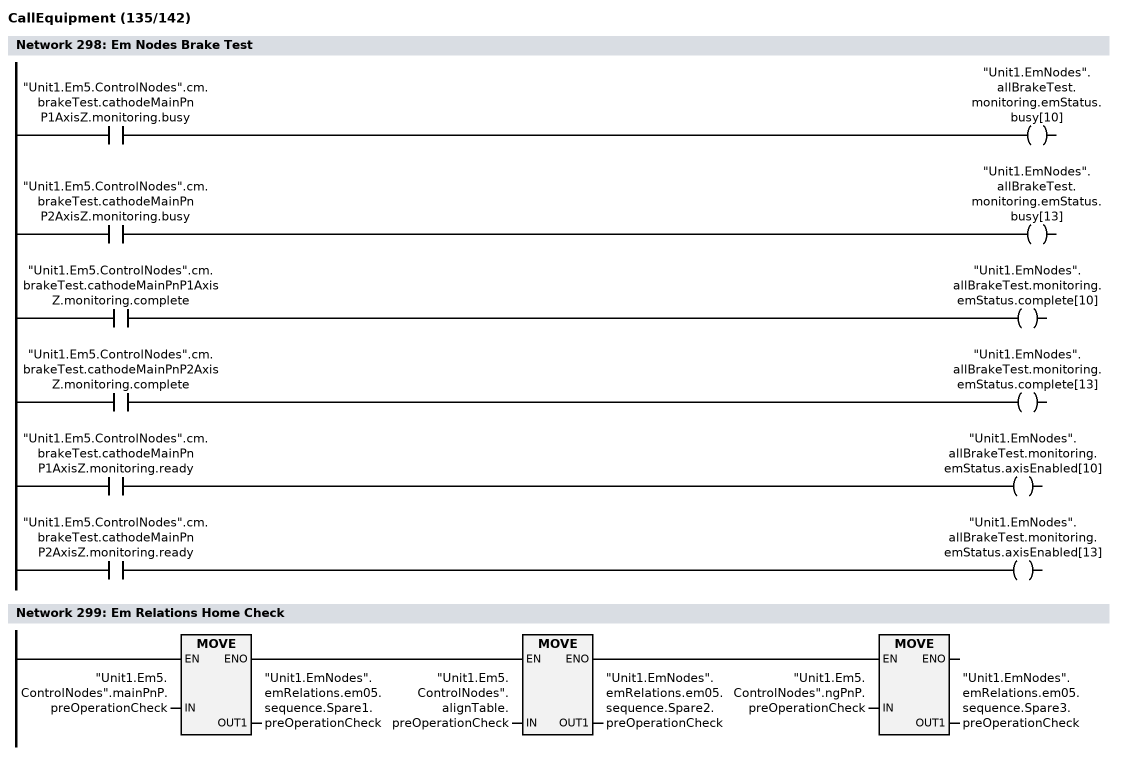
   RUNG wire#powerrail
      Contact( "Unit1.Em5.ControlNodes".cm.brakeTest.cathodeMainPnP1AxisZ.monitoring.busy )
      Coil( "Unit1.EmNodes".allBrakeTest.monitoring.emStatus.busy[10] )
   END_RUNG
   RUNG wire#powerrail
      Contact( "Unit1.Em5.ControlNodes".cm.brakeTest.cathodeMainPnP2AxisZ.monitoring.busy )
      Coil( "Unit1.EmNodes".allBrakeTest.monitoring.emStatus.busy[13] )
   END_RUNG
   RUNG wire#powerrail
      Contact( "Unit1.Em5.ControlNodes".cm.brakeTest.cathodeMainPnP1AxisZ.monitoring.complete )
      Coil( "Unit1.EmNodes".allBrakeTest.monitoring.emStatus.complete[10] )
   END_RUNG
   RUNG wire#powerrail
      Contact( "Unit1.Em5.ControlNodes".cm.brakeTest.cathodeMainPnP2AxisZ.monitoring.complete )
      Coil( "Unit1.EmNodes".allBrakeTest.monitoring.emStatus.complete[13] )
   END_RUNG
   RUNG wire#powerrail
      Contact( "Unit1.Em5.ControlNodes".cm.brakeTest.cathodeMainPnP1AxisZ.monitoring.ready )
      Coil( "Unit1.EmNodes".allBrakeTest.monitoring.emStatus.axisEnabled[10] )
   END_RUNG
   RUNG wire#powerrail
      Contact( "Unit1.Em5.ControlNodes".cm.brakeTest.cathodeMainPnP2AxisZ.monitoring.ready )
      Coil( "Unit1.EmNodes".allBrakeTest.monitoring.emStatus.axisEnabled[13] )
   END_RUNG
   // the same network as SCL:
   "Unit1.EmNodes".allBrakeTest.monitoring.emStatus.busy[10] := "Unit1.Em5.ControlNodes".cm.brakeTest.cathodeMainPnP1AxisZ.monitoring.busy;
   "Unit1.EmNodes".allBrakeTest.monitoring.emStatus.busy[13] := "Unit1.Em5.ControlNodes".cm.brakeTest.cathodeMainPnP2AxisZ.monitoring.busy;
   "Unit1.EmNodes".allBrakeTest.monitoring.emStatus.complete[10] := "Unit1.Em5.ControlNodes".cm.brakeTest.cathodeMainPnP1AxisZ.monitoring.complete;
   "Unit1.EmNodes".allBrakeTest.monitoring.emStatus.complete[13] := "Unit1.Em5.ControlNodes".cm.brakeTest.cathodeMainPnP2AxisZ.monitoring.complete;
   "Unit1.EmNodes".allBrakeTest.monitoring.emStatus.axisEnabled[10] := "Unit1.Em5.ControlNodes".cm.brakeTest.cathodeMainPnP1AxisZ.monitoring.ready;
   "Unit1.EmNodes".allBrakeTest.monitoring.emStatus.axisEnabled[13] := "Unit1.Em5.ControlNodes".cm.brakeTest.cathodeMainPnP2AxisZ.monitoring.ready;
END_REGION

REGION Network 299: Em Relations Home Check
   RUNG wire#powerrail
      Move(in := "Unit1.Em5.ControlNodes".mainPnP.preOperationCheck, out1 => "Unit1.EmNodes".emRelations.em05.sequence.Spare1.preOperationCheck)
      Move(in := "Unit1.Em5.ControlNodes".alignTable.preOperationCheck, out1 => "Unit1.EmNodes".emRelations.em05.sequence.Spare2.preOperationCheck)
      Move(in := "Unit1.Em5.ControlNodes".ngPnP.preOperationCheck, out1 => "Unit1.EmNodes".emRelations.em05.sequence.Spare3.preOperationCheck)
   END_RUNG
   // the same network as SCL:
   "Unit1.EmNodes".emRelations.em05.sequence.Spare1.preOperationCheck := "Unit1.Em5.ControlNodes".mainPnP.preOperationCheck;
   "Unit1.EmNodes".emRelations.em05.sequence.Spare2.preOperationCheck := "Unit1.Em5.ControlNodes".alignTable.preOperationCheck;
   "Unit1.EmNodes".emRelations.em05.sequence.Spare3.preOperationCheck := "Unit1.Em5.ControlNodes".ngPnP.preOperationCheck;
END_REGION

REGION Network 300: Em Relations Cylinder
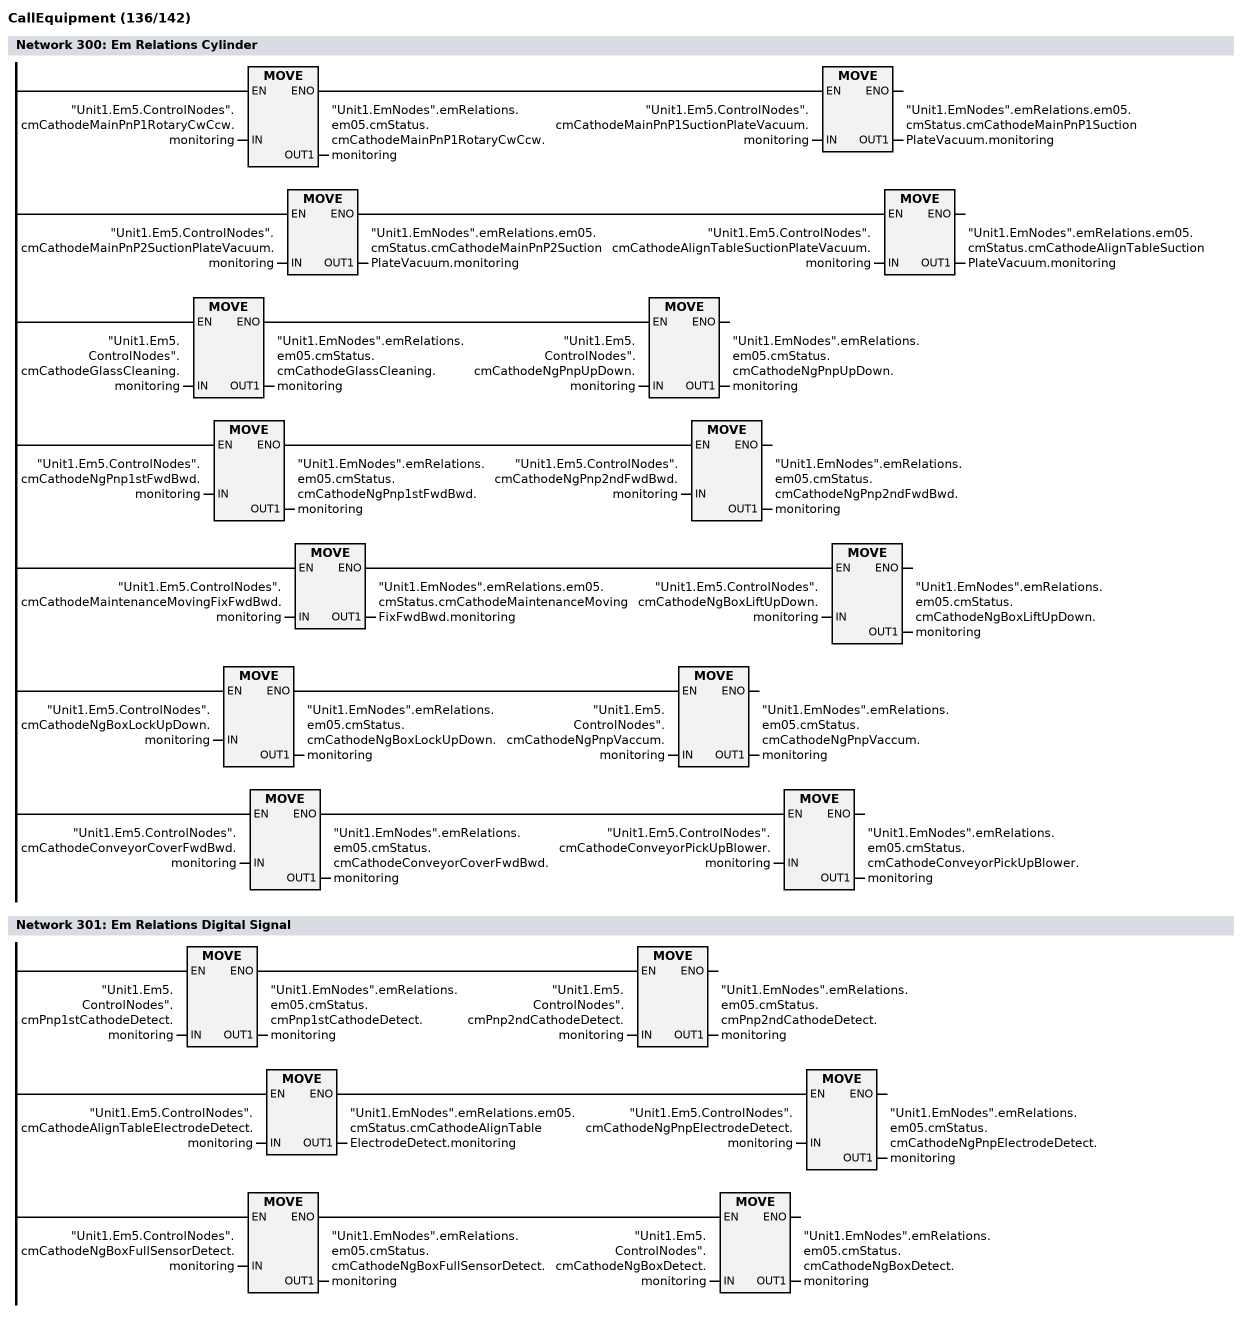
   RUNG wire#powerrail
      Move(in := "Unit1.Em5.ControlNodes".cmCathodeMainPnP1RotaryCwCcw.monitoring, out1 => "Unit1.EmNodes".emRelations.em05.cmStatus.cmCathodeMainPnP1RotaryCwCcw.monitoring)
      Move(in := "Unit1.Em5.ControlNodes".cmCathodeMainPnP1SuctionPlateVacuum.monitoring, out1 => "Unit1.EmNodes".emRelations.em05.cmStatus.cmCathodeMainPnP1SuctionPlateVacuum.monitoring)
   END_RUNG
   RUNG wire#powerrail
      Move(in := "Unit1.Em5.ControlNodes".cmCathodeMainPnP2SuctionPlateVacuum.monitoring, out1 => "Unit1.EmNodes".emRelations.em05.cmStatus.cmCathodeMainPnP2SuctionPlateVacuum.monitoring)
      Move(in := "Unit1.Em5.ControlNodes".cmCathodeAlignTableSuctionPlateVacuum.monitoring, out1 => "Unit1.EmNodes".emRelations.em05.cmStatus.cmCathodeAlignTableSuctionPlateVacuum.monitoring)
   END_RUNG
   RUNG wire#powerrail
      Move(in := "Unit1.Em5.ControlNodes".cmCathodeGlassCleaning.monitoring, out1 => "Unit1.EmNodes".emRelations.em05.cmStatus.cmCathodeGlassCleaning.monitoring)
      Move(in := "Unit1.Em5.ControlNodes".cmCathodeNgPnpUpDown.monitoring, out1 => "Unit1.EmNodes".emRelations.em05.cmStatus.cmCathodeNgPnpUpDown.monitoring)
   END_RUNG
   RUNG wire#powerrail
      Move(in := "Unit1.Em5.ControlNodes".cmCathodeNgPnp1stFwdBwd.monitoring, out1 => "Unit1.EmNodes".emRelations.em05.cmStatus.cmCathodeNgPnp1stFwdBwd.monitoring)
      Move(in := "Unit1.Em5.ControlNodes".cmCathodeNgPnp2ndFwdBwd.monitoring, out1 => "Unit1.EmNodes".emRelations.em05.cmStatus.cmCathodeNgPnp2ndFwdBwd.monitoring)
   END_RUNG
   RUNG wire#powerrail
      Move(in := "Unit1.Em5.ControlNodes".cmCathodeMaintenanceMovingFixFwdBwd.monitoring, out1 => "Unit1.EmNodes".emRelations.em05.cmStatus.cmCathodeMaintenanceMovingFixFwdBwd.monitoring)
      Move(in := "Unit1.Em5.ControlNodes".cmCathodeNgBoxLiftUpDown.monitoring, out1 => "Unit1.EmNodes".emRelations.em05.cmStatus.cmCathodeNgBoxLiftUpDown.monitoring)
   END_RUNG
   RUNG wire#powerrail
      Move(in := "Unit1.Em5.ControlNodes".cmCathodeNgBoxLockUpDown.monitoring, out1 => "Unit1.EmNodes".emRelations.em05.cmStatus.cmCathodeNgBoxLockUpDown.monitoring)
      Move(in := "Unit1.Em5.ControlNodes".cmCathodeNgPnpVaccum.monitoring, out1 => "Unit1.EmNodes".emRelations.em05.cmStatus.cmCathodeNgPnpVaccum.monitoring)
   END_RUNG
   RUNG wire#powerrail
      Move(in := "Unit1.Em5.ControlNodes".cmCathodeConveyorCoverFwdBwd.monitoring, out1 => "Unit1.EmNodes".emRelations.em05.cmStatus.cmCathodeConveyorCoverFwdBwd.monitoring)
      Move(in := "Unit1.Em5.ControlNodes".cmCathodeConveyorPickUpBlower.monitoring, out1 => "Unit1.EmNodes".emRelations.em05.cmStatus.cmCathodeConveyorPickUpBlower.monitoring)
   END_RUNG
   // the same network as SCL:
   "Unit1.EmNodes".emRelations.em05.cmStatus.cmCathodeMainPnP1RotaryCwCcw.monitoring := "Unit1.Em5.ControlNodes".cmCathodeMainPnP1RotaryCwCcw.monitoring;
   "Unit1.EmNodes".emRelations.em05.cmStatus.cmCathodeMainPnP1SuctionPlateVacuum.monitoring := "Unit1.Em5.ControlNodes".cmCathodeMainPnP1SuctionPlateVacuum.monitoring;
   "Unit1.EmNodes".emRelations.em05.cmStatus.cmCathodeMainPnP2SuctionPlateVacuum.monitoring := "Unit1.Em5.ControlNodes".cmCathodeMainPnP2SuctionPlateVacuum.monitoring;
   "Unit1.EmNodes".emRelations.em05.cmStatus.cmCathodeAlignTableSuctionPlateVacuum.monitoring := "Unit1.Em5.ControlNodes".cmCathodeAlignTableSuctionPlateVacuum.monitoring;
   "Unit1.EmNodes".emRelations.em05.cmStatus.cmCathodeGlassCleaning.monitoring := "Unit1.Em5.ControlNodes".cmCathodeGlassCleaning.monitoring;
   "Unit1.EmNodes".emRelations.em05.cmStatus.cmCathodeNgPnpUpDown.monitoring := "Unit1.Em5.ControlNodes".cmCathodeNgPnpUpDown.monitoring;
   "Unit1.EmNodes".emRelations.em05.cmStatus.cmCathodeNgPnp1stFwdBwd.monitoring := "Unit1.Em5.ControlNodes".cmCathodeNgPnp1stFwdBwd.monitoring;
   "Unit1.EmNodes".emRelations.em05.cmStatus.cmCathodeNgPnp2ndFwdBwd.monitoring := "Unit1.Em5.ControlNodes".cmCathodeNgPnp2ndFwdBwd.monitoring;
   "Unit1.EmNodes".emRelations.em05.cmStatus.cmCathodeMaintenanceMovingFixFwdBwd.monitoring := "Unit1.Em5.ControlNodes".cmCathodeMaintenanceMovingFixFwdBwd.monitoring;
   "Unit1.EmNodes".emRelations.em05.cmStatus.cmCathodeNgBoxLiftUpDown.monitoring := "Unit1.Em5.ControlNodes".cmCathodeNgBoxLiftUpDown.monitoring;
   "Unit1.EmNodes".emRelations.em05.cmStatus.cmCathodeNgBoxLockUpDown.monitoring := "Unit1.Em5.ControlNodes".cmCathodeNgBoxLockUpDown.monitoring;
   "Unit1.EmNodes".emRelations.em05.cmStatus.cmCathodeNgPnpVaccum.monitoring := "Unit1.Em5.ControlNodes".cmCathodeNgPnpVaccum.monitoring;
   "Unit1.EmNodes".emRelations.em05.cmStatus.cmCathodeConveyorCoverFwdBwd.monitoring := "Unit1.Em5.ControlNodes".cmCathodeConveyorCoverFwdBwd.monitoring;
   "Unit1.EmNodes".emRelations.em05.cmStatus.cmCathodeConveyorPickUpBlower.monitoring := "Unit1.Em5.ControlNodes".cmCathodeConveyorPickUpBlower.monitoring;
END_REGION

REGION Network 301: Em Relations Digital Signal
   RUNG wire#powerrail
      Move(in := "Unit1.Em5.ControlNodes".cmPnp1stCathodeDetect.monitoring, out1 => "Unit1.EmNodes".emRelations.em05.cmStatus.cmPnp1stCathodeDetect.monitoring)
      Move(in := "Unit1.Em5.ControlNodes".cmPnp2ndCathodeDetect.monitoring, out1 => "Unit1.EmNodes".emRelations.em05.cmStatus.cmPnp2ndCathodeDetect.monitoring)
   END_RUNG
   RUNG wire#powerrail
      Move(in := "Unit1.Em5.ControlNodes".cmCathodeAlignTableElectrodeDetect.monitoring, out1 => "Unit1.EmNodes".emRelations.em05.cmStatus.cmCathodeAlignTableElectrodeDetect.monitoring)
      Move(in := "Unit1.Em5.ControlNodes".cmCathodeNgPnpElectrodeDetect.monitoring, out1 => "Unit1.EmNodes".emRelations.em05.cmStatus.cmCathodeNgPnpElectrodeDetect.monitoring)
   END_RUNG
   RUNG wire#powerrail
      Move(in := "Unit1.Em5.ControlNodes".cmCathodeNgBoxFullSensorDetect.monitoring, out1 => "Unit1.EmNodes".emRelations.em05.cmStatus.cmCathodeNgBoxFullSensorDetect.monitoring)
      Move(in := "Unit1.Em5.ControlNodes".cmCathodeNgBoxDetect.monitoring, out1 => "Unit1.EmNodes".emRelations.em05.cmStatus.cmCathodeNgBoxDetect.monitoring)
   END_RUNG
   // the same network as SCL:
   "Unit1.EmNodes".emRelations.em05.cmStatus.cmPnp1stCathodeDetect.monitoring := "Unit1.Em5.ControlNodes".cmPnp1stCathodeDetect.monitoring;
   "Unit1.EmNodes".emRelations.em05.cmStatus.cmPnp2ndCathodeDetect.monitoring := "Unit1.Em5.ControlNodes".cmPnp2ndCathodeDetect.monitoring;
   "Unit1.EmNodes".emRelations.em05.cmStatus.cmCathodeAlignTableElectrodeDetect.monitoring := "Unit1.Em5.ControlNodes".cmCathodeAlignTableElectrodeDetect.monitoring;
   "Unit1.EmNodes".emRelations.em05.cmStatus.cmCathodeNgPnpElectrodeDetect.monitoring := "Unit1.Em5.ControlNodes".cmCathodeNgPnpElectrodeDetect.monitoring;
   "Unit1.EmNodes".emRelations.em05.cmStatus.cmCathodeNgBoxFullSensorDetect.monitoring := "Unit1.Em5.ControlNodes".cmCathodeNgBoxFullSensorDetect.monitoring;
   "Unit1.EmNodes".emRelations.em05.cmStatus.cmCathodeNgBoxDetect.monitoring := "Unit1.Em5.ControlNodes".cmCathodeNgBoxDetect.monitoring;
END_REGION

REGION Network 302: Em Relations Select Job Status
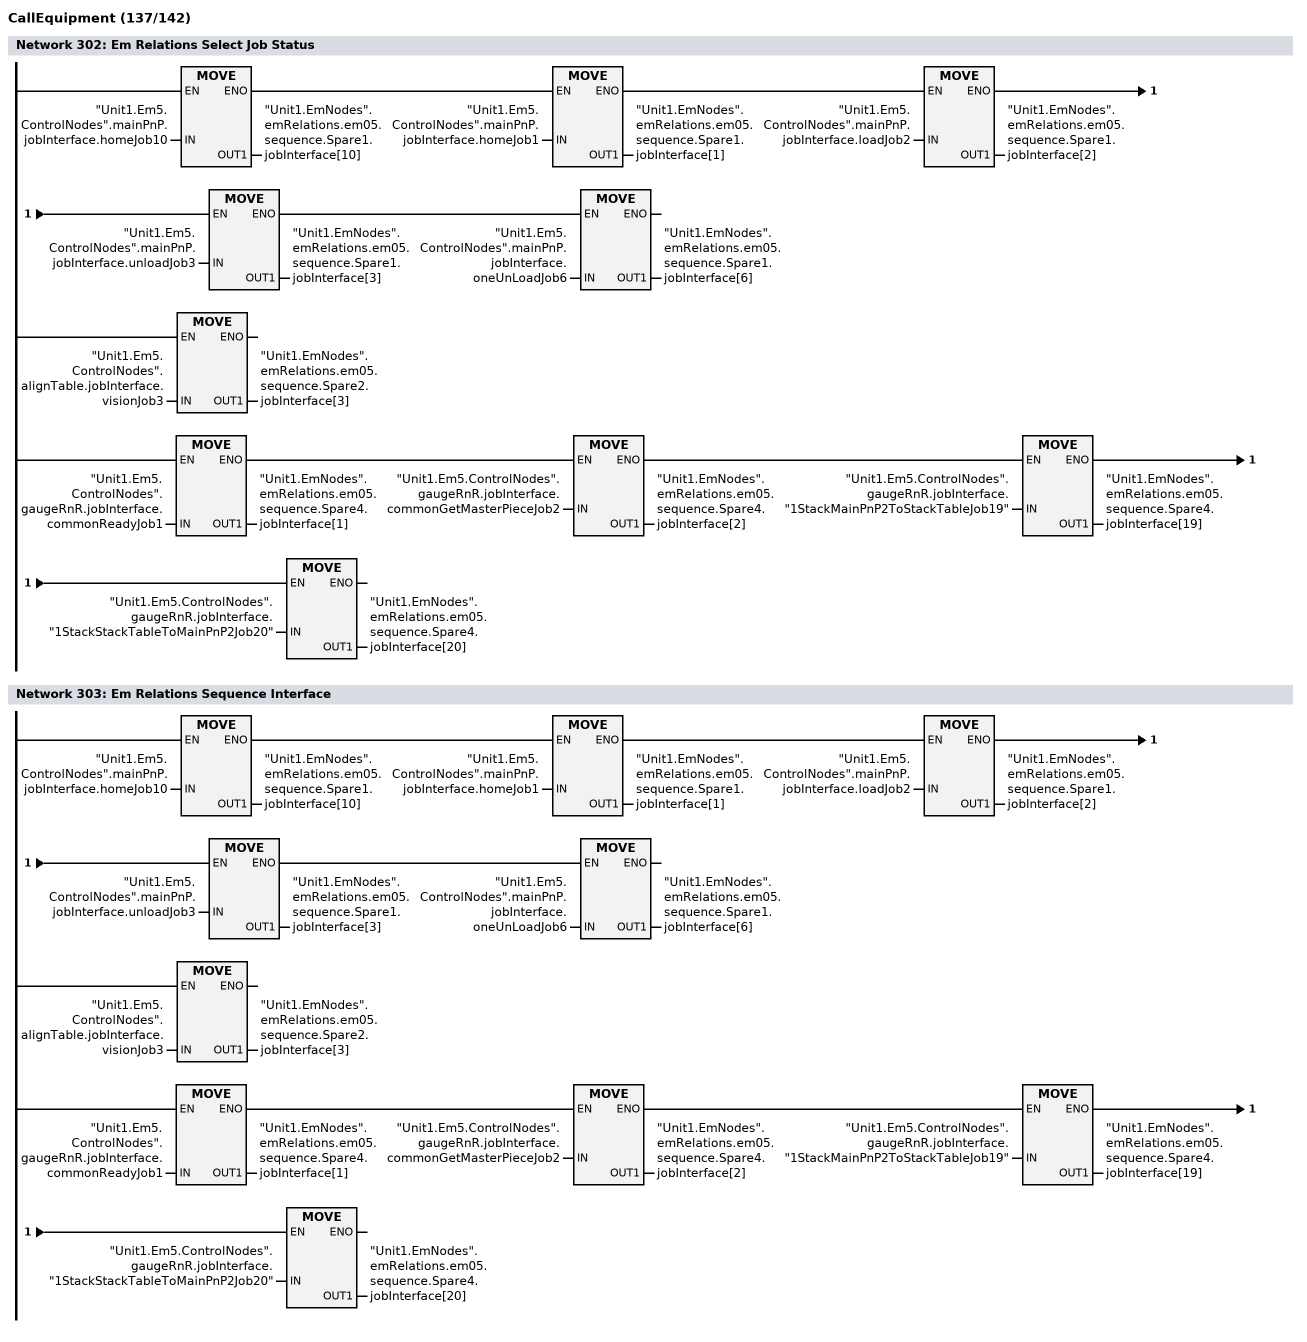
   RUNG wire#powerrail
      Move(in := "Unit1.Em5.ControlNodes".mainPnP.jobInterface.homeJob10, out1 => "Unit1.EmNodes".emRelations.em05.sequence.Spare1.jobInterface[10])
      Move(in := "Unit1.Em5.ControlNodes".mainPnP.jobInterface.homeJob1, out1 => "Unit1.EmNodes".emRelations.em05.sequence.Spare1.jobInterface[1])
      Move(in := "Unit1.Em5.ControlNodes".mainPnP.jobInterface.loadJob2, out1 => "Unit1.EmNodes".emRelations.em05.sequence.Spare1.jobInterface[2])
      Move(in := "Unit1.Em5.ControlNodes".mainPnP.jobInterface.unloadJob3, out1 => "Unit1.EmNodes".emRelations.em05.sequence.Spare1.jobInterface[3])
      Move(in := "Unit1.Em5.ControlNodes".mainPnP.jobInterface.oneUnLoadJob6, out1 => "Unit1.EmNodes".emRelations.em05.sequence.Spare1.jobInterface[6])
   END_RUNG
   RUNG wire#powerrail
      Move(in := "Unit1.Em5.ControlNodes".alignTable.jobInterface.visionJob3, out1 => "Unit1.EmNodes".emRelations.em05.sequence.Spare2.jobInterface[3])
   END_RUNG
   RUNG wire#powerrail
      Move(in := "Unit1.Em5.ControlNodes".gaugeRnR.jobInterface.commonReadyJob1, out1 => "Unit1.EmNodes".emRelations.em05.sequence.Spare4.jobInterface[1])
      Move(in := "Unit1.Em5.ControlNodes".gaugeRnR.jobInterface.commonGetMasterPieceJob2, out1 => "Unit1.EmNodes".emRelations.em05.sequence.Spare4.jobInterface[2])
      Move(in := "Unit1.Em5.ControlNodes".gaugeRnR.jobInterface."1StackMainPnP2ToStackTableJob19", out1 => "Unit1.EmNodes".emRelations.em05.sequence.Spare4.jobInterface[19])
      Move(in := "Unit1.Em5.ControlNodes".gaugeRnR.jobInterface."1StackStackTableToMainPnP2Job20", out1 => "Unit1.EmNodes".emRelations.em05.sequence.Spare4.jobInterface[20])
   END_RUNG
   // the same network as SCL:
   "Unit1.EmNodes".emRelations.em05.sequence.Spare1.jobInterface[10] := "Unit1.Em5.ControlNodes".mainPnP.jobInterface.homeJob10;
   "Unit1.EmNodes".emRelations.em05.sequence.Spare1.jobInterface[1] := "Unit1.Em5.ControlNodes".mainPnP.jobInterface.homeJob1;
   "Unit1.EmNodes".emRelations.em05.sequence.Spare1.jobInterface[2] := "Unit1.Em5.ControlNodes".mainPnP.jobInterface.loadJob2;
   "Unit1.EmNodes".emRelations.em05.sequence.Spare1.jobInterface[3] := "Unit1.Em5.ControlNodes".mainPnP.jobInterface.unloadJob3;
   "Unit1.EmNodes".emRelations.em05.sequence.Spare1.jobInterface[6] := "Unit1.Em5.ControlNodes".mainPnP.jobInterface.oneUnLoadJob6;
   "Unit1.EmNodes".emRelations.em05.sequence.Spare2.jobInterface[3] := "Unit1.Em5.ControlNodes".alignTable.jobInterface.visionJob3;
   "Unit1.EmNodes".emRelations.em05.sequence.Spare4.jobInterface[1] := "Unit1.Em5.ControlNodes".gaugeRnR.jobInterface.commonReadyJob1;
   "Unit1.EmNodes".emRelations.em05.sequence.Spare4.jobInterface[2] := "Unit1.Em5.ControlNodes".gaugeRnR.jobInterface.commonGetMasterPieceJob2;
   "Unit1.EmNodes".emRelations.em05.sequence.Spare4.jobInterface[19] := "Unit1.Em5.ControlNodes".gaugeRnR.jobInterface."1StackMainPnP2ToStackTableJob19";
   "Unit1.EmNodes".emRelations.em05.sequence.Spare4.jobInterface[20] := "Unit1.Em5.ControlNodes".gaugeRnR.jobInterface."1StackStackTableToMainPnP2Job20";
END_REGION

REGION Network 303: Em Relations Sequence Interface
   RUNG wire#powerrail
      Move(in := "Unit1.Em5.ControlNodes".mainPnP.jobInterface.homeJob10, out1 => "Unit1.EmNodes".emRelations.em05.sequence.Spare1.jobInterface[10])
      Move(in := "Unit1.Em5.ControlNodes".mainPnP.jobInterface.homeJob1, out1 => "Unit1.EmNodes".emRelations.em05.sequence.Spare1.jobInterface[1])
      Move(in := "Unit1.Em5.ControlNodes".mainPnP.jobInterface.loadJob2, out1 => "Unit1.EmNodes".emRelations.em05.sequence.Spare1.jobInterface[2])
      Move(in := "Unit1.Em5.ControlNodes".mainPnP.jobInterface.unloadJob3, out1 => "Unit1.EmNodes".emRelations.em05.sequence.Spare1.jobInterface[3])
      Move(in := "Unit1.Em5.ControlNodes".mainPnP.jobInterface.oneUnLoadJob6, out1 => "Unit1.EmNodes".emRelations.em05.sequence.Spare1.jobInterface[6])
   END_RUNG
   RUNG wire#powerrail
      Move(in := "Unit1.Em5.ControlNodes".alignTable.jobInterface.visionJob3, out1 => "Unit1.EmNodes".emRelations.em05.sequence.Spare2.jobInterface[3])
   END_RUNG
   RUNG wire#powerrail
      Move(in := "Unit1.Em5.ControlNodes".gaugeRnR.jobInterface.commonReadyJob1, out1 => "Unit1.EmNodes".emRelations.em05.sequence.Spare4.jobInterface[1])
      Move(in := "Unit1.Em5.ControlNodes".gaugeRnR.jobInterface.commonGetMasterPieceJob2, out1 => "Unit1.EmNodes".emRelations.em05.sequence.Spare4.jobInterface[2])
      Move(in := "Unit1.Em5.ControlNodes".gaugeRnR.jobInterface."1StackMainPnP2ToStackTableJob19", out1 => "Unit1.EmNodes".emRelations.em05.sequence.Spare4.jobInterface[19])
      Move(in := "Unit1.Em5.ControlNodes".gaugeRnR.jobInterface."1StackStackTableToMainPnP2Job20", out1 => "Unit1.EmNodes".emRelations.em05.sequence.Spare4.jobInterface[20])
   END_RUNG
   // the same network as SCL:
   "Unit1.EmNodes".emRelations.em05.sequence.Spare1.jobInterface[10] := "Unit1.Em5.ControlNodes".mainPnP.jobInterface.homeJob10;
   "Unit1.EmNodes".emRelations.em05.sequence.Spare1.jobInterface[1] := "Unit1.Em5.ControlNodes".mainPnP.jobInterface.homeJob1;
   "Unit1.EmNodes".emRelations.em05.sequence.Spare1.jobInterface[2] := "Unit1.Em5.ControlNodes".mainPnP.jobInterface.loadJob2;
   "Unit1.EmNodes".emRelations.em05.sequence.Spare1.jobInterface[3] := "Unit1.Em5.ControlNodes".mainPnP.jobInterface.unloadJob3;
   "Unit1.EmNodes".emRelations.em05.sequence.Spare1.jobInterface[6] := "Unit1.Em5.ControlNodes".mainPnP.jobInterface.oneUnLoadJob6;
   "Unit1.EmNodes".emRelations.em05.sequence.Spare2.jobInterface[3] := "Unit1.Em5.ControlNodes".alignTable.jobInterface.visionJob3;
   "Unit1.EmNodes".emRelations.em05.sequence.Spare4.jobInterface[1] := "Unit1.Em5.ControlNodes".gaugeRnR.jobInterface.commonReadyJob1;
   "Unit1.EmNodes".emRelations.em05.sequence.Spare4.jobInterface[2] := "Unit1.Em5.ControlNodes".gaugeRnR.jobInterface.commonGetMasterPieceJob2;
   "Unit1.EmNodes".emRelations.em05.sequence.Spare4.jobInterface[19] := "Unit1.Em5.ControlNodes".gaugeRnR.jobInterface."1StackMainPnP2ToStackTableJob19";
   "Unit1.EmNodes".emRelations.em05.sequence.Spare4.jobInterface[20] := "Unit1.Em5.ControlNodes".gaugeRnR.jobInterface."1StackStackTableToMainPnP2Job20";
END_REGION

REGION Network 304: Em Relations Softcam
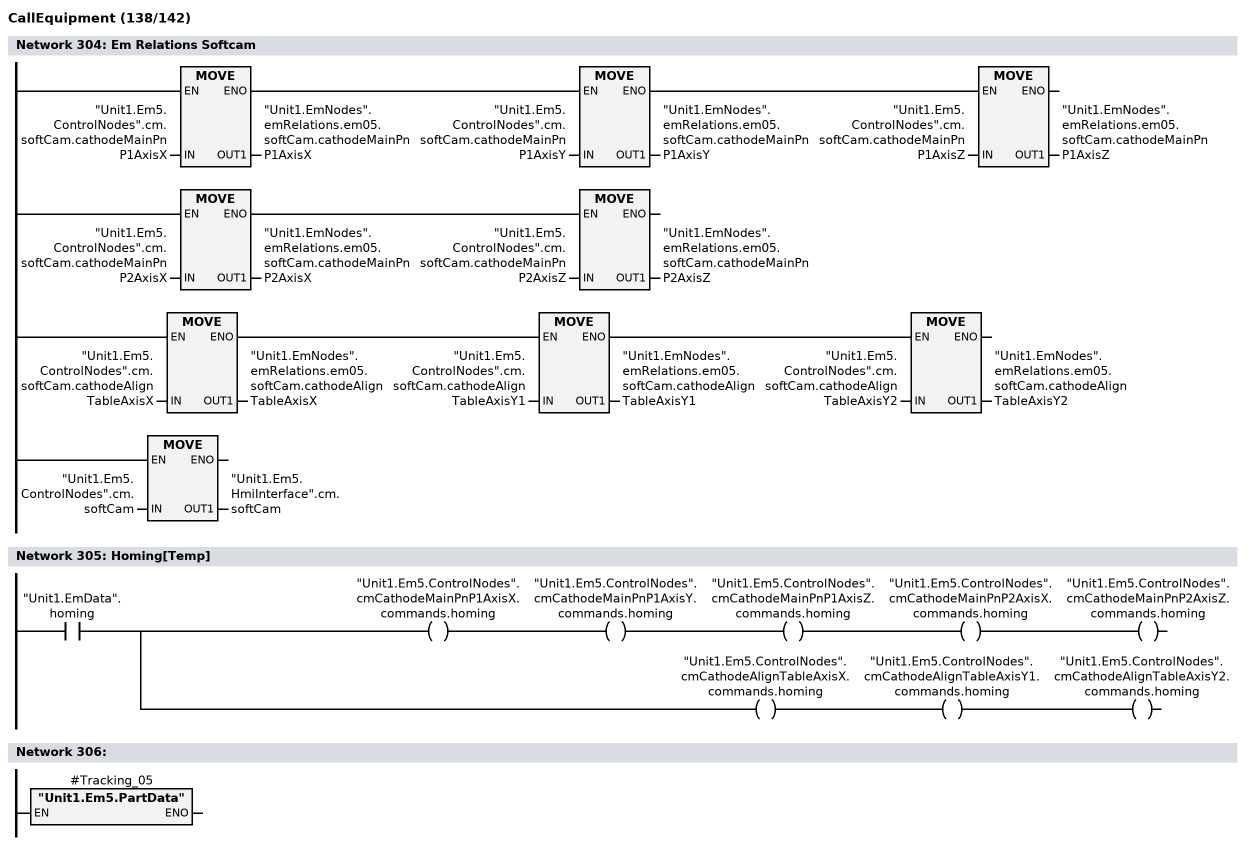
   RUNG wire#powerrail
      Move(in := "Unit1.Em5.ControlNodes".cm.softCam.cathodeMainPnP1AxisX, out1 => "Unit1.EmNodes".emRelations.em05.softCam.cathodeMainPnP1AxisX)
      Move(in := "Unit1.Em5.ControlNodes".cm.softCam.cathodeMainPnP1AxisY, out1 => "Unit1.EmNodes".emRelations.em05.softCam.cathodeMainPnP1AxisY)
      Move(in := "Unit1.Em5.ControlNodes".cm.softCam.cathodeMainPnP1AxisZ, out1 => "Unit1.EmNodes".emRelations.em05.softCam.cathodeMainPnP1AxisZ)
   END_RUNG
   RUNG wire#powerrail
      Move(in := "Unit1.Em5.ControlNodes".cm.softCam.cathodeMainPnP2AxisX, out1 => "Unit1.EmNodes".emRelations.em05.softCam.cathodeMainPnP2AxisX)
      Move(in := "Unit1.Em5.ControlNodes".cm.softCam.cathodeMainPnP2AxisZ, out1 => "Unit1.EmNodes".emRelations.em05.softCam.cathodeMainPnP2AxisZ)
   END_RUNG
   RUNG wire#powerrail
      Move(in := "Unit1.Em5.ControlNodes".cm.softCam.cathodeAlignTableAxisX, out1 => "Unit1.EmNodes".emRelations.em05.softCam.cathodeAlignTableAxisX)
      Move(in := "Unit1.Em5.ControlNodes".cm.softCam.cathodeAlignTableAxisY1, out1 => "Unit1.EmNodes".emRelations.em05.softCam.cathodeAlignTableAxisY1)
      Move(in := "Unit1.Em5.ControlNodes".cm.softCam.cathodeAlignTableAxisY2, out1 => "Unit1.EmNodes".emRelations.em05.softCam.cathodeAlignTableAxisY2)
   END_RUNG
   RUNG wire#powerrail
      Move(in := "Unit1.Em5.ControlNodes".cm.softCam, out1 => "Unit1.Em5.HmiInterface".cm.softCam)
   END_RUNG
   // the same network as SCL:
   "Unit1.EmNodes".emRelations.em05.softCam.cathodeMainPnP1AxisX := "Unit1.Em5.ControlNodes".cm.softCam.cathodeMainPnP1AxisX;
   "Unit1.EmNodes".emRelations.em05.softCam.cathodeMainPnP1AxisY := "Unit1.Em5.ControlNodes".cm.softCam.cathodeMainPnP1AxisY;
   "Unit1.EmNodes".emRelations.em05.softCam.cathodeMainPnP1AxisZ := "Unit1.Em5.ControlNodes".cm.softCam.cathodeMainPnP1AxisZ;
   "Unit1.EmNodes".emRelations.em05.softCam.cathodeMainPnP2AxisX := "Unit1.Em5.ControlNodes".cm.softCam.cathodeMainPnP2AxisX;
   "Unit1.EmNodes".emRelations.em05.softCam.cathodeMainPnP2AxisZ := "Unit1.Em5.ControlNodes".cm.softCam.cathodeMainPnP2AxisZ;
   "Unit1.EmNodes".emRelations.em05.softCam.cathodeAlignTableAxisX := "Unit1.Em5.ControlNodes".cm.softCam.cathodeAlignTableAxisX;
   "Unit1.EmNodes".emRelations.em05.softCam.cathodeAlignTableAxisY1 := "Unit1.Em5.ControlNodes".cm.softCam.cathodeAlignTableAxisY1;
   "Unit1.EmNodes".emRelations.em05.softCam.cathodeAlignTableAxisY2 := "Unit1.Em5.ControlNodes".cm.softCam.cathodeAlignTableAxisY2;
   "Unit1.Em5.HmiInterface".cm.softCam := "Unit1.Em5.ControlNodes".cm.softCam;
END_REGION

REGION Network 305: Homing[Temp]
   RUNG wire#powerrail
      Contact( "Unit1.EmData".homing )
      wire#w1
      Coil( "Unit1.Em5.ControlNodes".cmCathodeMainPnP1AxisX.commands.homing )
      Coil( "Unit1.Em5.ControlNodes".cmCathodeMainPnP1AxisY.commands.homing )
      Coil( "Unit1.Em5.ControlNodes".cmCathodeMainPnP1AxisZ.commands.homing )
      Coil( "Unit1.Em5.ControlNodes".cmCathodeMainPnP2AxisX.commands.homing )
      Coil( "Unit1.Em5.ControlNodes".cmCathodeMainPnP2AxisZ.commands.homing )
   END_RUNG
   RUNG wire#w1
      Coil( "Unit1.Em5.ControlNodes".cmCathodeAlignTableAxisX.commands.homing )
      Coil( "Unit1.Em5.ControlNodes".cmCathodeAlignTableAxisY1.commands.homing )
      Coil( "Unit1.Em5.ControlNodes".cmCathodeAlignTableAxisY2.commands.homing )
   END_RUNG
   // the same network as SCL:
   "Unit1.Em5.ControlNodes".cmCathodeMainPnP1AxisX.commands.homing := "Unit1.EmData".homing;
   "Unit1.Em5.ControlNodes".cmCathodeMainPnP1AxisY.commands.homing := "Unit1.EmData".homing;
   "Unit1.Em5.ControlNodes".cmCathodeMainPnP1AxisZ.commands.homing := "Unit1.EmData".homing;
   "Unit1.Em5.ControlNodes".cmCathodeMainPnP2AxisX.commands.homing := "Unit1.EmData".homing;
   "Unit1.Em5.ControlNodes".cmCathodeMainPnP2AxisZ.commands.homing := "Unit1.EmData".homing;
   "Unit1.Em5.ControlNodes".cmCathodeAlignTableAxisX.commands.homing := "Unit1.EmData".homing;
   "Unit1.Em5.ControlNodes".cmCathodeAlignTableAxisY1.commands.homing := "Unit1.EmData".homing;
   "Unit1.Em5.ControlNodes".cmCathodeAlignTableAxisY2.commands.homing := "Unit1.EmData".homing;
END_REGION

REGION Network 306
   RUNG wire#powerrail
      #Tracking_05()
   END_RUNG
   // the same network as SCL:
   #Tracking_05();   // "Unit1.Em5.PartData"
END_REGION

REGION Network 307 (SCL): SyncMotion Configuration
   "Unit1.MotionNodes".PLCToMotion.TechnologyObject.Axis.CathodePnPX1 := "Unit1.Em5.Config".axis[1];
   "Unit1.MotionNodes".PLCToMotion.TechnologyObject.Axis.CathodePnPX2 := "Unit1.Em5.Config".axis[2];
   "Unit1.MotionNodes".PLCToMotion.TechnologyObject.Axis.CathodePnPZ1 := "Unit1.Em5.Config".axis[4];
   "Unit1.MotionNodes".PLCToMotion.TechnologyObject.Axis.CathodePnPZ2 := "Unit1.Em5.Config".axis[5];

   // _.Unit1.SyncMotion.Configuration.TechnologyObjects.StackMain.Cam.CathodePnPX1Cam := Config.cam[1];
   // _.Unit1.SyncMotion.Configuration.TechnologyObjects.StackMain.Cam.CathodePnPX2Cam := Config.cam[2];
   // _.Unit1.SyncMotion.Configuration.TechnologyObjects.StackMain.Cam.CathodePnPZ1Cam := Config.cam[3];
   // _.Unit1.SyncMotion.Configuration.TechnologyObjects.StackMain.Cam.CathodePnPZ2Cam := Config.cam[4];

   "Unit1.Em5.Config".outputCam[1] := "CathodePnP1XFwd";
   "Unit1.Em5.Config".outputCam[2] := "CathodePnP1XBwd";
   "Unit1.Em5.Config".outputCam[3] := "CathodePnP2XFwd";
   "Unit1.Em5.Config".outputCam[4] := "CathodePnP2XBwd";
   "Unit1.Em5.Config".outputCam[5] := "CathodePnPZ1Down1";
   "Unit1.Em5.Config".outputCam[6] := "CathodePnPZ1Up1";
   "Unit1.Em5.Config".outputCam[7] := "CathodePnPZ2Down1";
   "Unit1.Em5.Config".outputCam[8] := "CathodePnPZ2Up1";
   "Unit1.Em5.Config".outputCam[9] := "CathodePnPZ1Down2";
   "Unit1.Em5.Config".outputCam[10] := "CathodePnPZ1Up2";
   "Unit1.Em5.Config".outputCam[11] := "CathodePnPZ2Down2";
   "Unit1.Em5.Config".outputCam[12] := "CathodePnPZ2Up2";
   "Unit1.Em5.Config".outputCam[13] := "CathodePnPZ1SuctionOn";
   "Unit1.Em5.Config".outputCam[14] := "CathodePnPZ1SuctionOff";
   "Unit1.Em5.Config".outputCam[15] := "CathodePnPZ1ReelCutBlow";
   "Unit1.Em5.Config".outputCam[16] := "CathodePnPZ2SuctionOn";
   "Unit1.Em5.Config".outputCam[17] := "CathodePnPZ2SuctionOff";
   "Unit1.Em5.Config".outputCam[18] := "CathodeAlignSuctionOn";
   "Unit1.Em5.Config".outputCam[19] := "CathodeAlignSuctionOff";
   "Unit1.Em5.Config".outputCam[20] := "CathodePnPZ1ReelCutDataDeleteOn";
   "Unit1.Em5.Config".outputCam[21] := "CathodePnP1XReelCutDataDeleteOff";
   "Unit1.Em5.Config".outputCam[22] := "CathodeAlignVision";


   "Unit1.MotionNodes".PLCToMotion.TechnologyObject.OutputCam.CathodePnPX1BwdOutputCam := "Unit1.Em5.Config".outputCam[1];
   "Unit1.MotionNodes".PLCToMotion.TechnologyObject.OutputCam.CathodePnPX1FwdOutputCam := "Unit1.Em5.Config".outputCam[2];
   "Unit1.MotionNodes".PLCToMotion.TechnologyObject.OutputCam.CathodePnPX2BwdOutputCam := "Unit1.Em5.Config".outputCam[3];
   "Unit1.MotionNodes".PLCToMotion.TechnologyObject.OutputCam.CathodePnPX2FwdOutputCam := "Unit1.Em5.Config".outputCam[4];
   "Unit1.MotionNodes".PLCToMotion.TechnologyObject.OutputCam.CathodePnPZ1Down1OutputCam := "Unit1.Em5.Config".outputCam[5];
   "Unit1.MotionNodes".PLCToMotion.TechnologyObject.OutputCam.CathodePnPZ1Up1OutputCam := "Unit1.Em5.Config".outputCam[6];
   "Unit1.MotionNodes".PLCToMotion.TechnologyObject.OutputCam.CathodePnPZ2Down1OutputCam := "Unit1.Em5.Config".outputCam[7];
   "Unit1.MotionNodes".PLCToMotion.TechnologyObject.OutputCam.CathodePnPZ2Up1OutputCam := "Unit1.Em5.Config".outputCam[8];
   "Unit1.MotionNodes".PLCToMotion.TechnologyObject.OutputCam.CathodePnPZ1Down2OutputCam := "Unit1.Em5.Config".outputCam[9];
   "Unit1.MotionNodes".PLCToMotion.TechnologyObject.OutputCam.CathodePnPZ1Up2OutputCam := "Unit1.Em5.Config".outputCam[10];
   "Unit1.MotionNodes".PLCToMotion.TechnologyObject.OutputCam.CathodePnPZ2Down2OutputCam := "Unit1.Em5.Config".outputCam[11];
   "Unit1.MotionNodes".PLCToMotion.TechnologyObject.OutputCam.CathodePnPZ2Up2OutputCam := "Unit1.Em5.Config".outputCam[12];
   "Unit1.MotionNodes".PLCToMotion.TechnologyObject.OutputCam.CathodePnPZ1SuctionOnOutputCam := "Unit1.Em5.Config".outputCam[13];
   "Unit1.MotionNodes".PLCToMotion.TechnologyObject.OutputCam.CathodePnPZ1SuctionOffOutputCam := "Unit1.Em5.Config".outputCam[14];
   "Unit1.MotionNodes".PLCToMotion.TechnologyObject.OutputCam.CathodePnPZ1ReelCutBlowOutputCam := "Unit1.Em5.Config".outputCam[15];
   "Unit1.MotionNodes".PLCToMotion.TechnologyObject.OutputCam.CathodePnPZ2SuctionOnOutputCam := "Unit1.Em5.Config".outputCam[16];
   "Unit1.MotionNodes".PLCToMotion.TechnologyObject.OutputCam.CathodePnPZ2SuctionOffOutputCam := "Unit1.Em5.Config".outputCam[17];
   "Unit1.MotionNodes".PLCToMotion.TechnologyObject.OutputCam.CathodeAlignSuctionOnOutputCam := "Unit1.Em5.Config".outputCam[18];
   "Unit1.MotionNodes".PLCToMotion.TechnologyObject.OutputCam.CathodeAlignSuctionOffOutputCam := "Unit1.Em5.Config".outputCam[19];
   "Unit1.MotionNodes".PLCToMotion.TechnologyObject.OutputCam.CathodePnPZ1ReelCutDataDeleteOnOutputCam := "Unit1.Em5.Config".outputCam[20];
   "Unit1.MotionNodes".PLCToMotion.TechnologyObject.OutputCam.CathodePnP1XReelCutDataDeleteOffOutputCam := "Unit1.Em5.Config".outputCam[21];
   "Unit1.MotionNodes".PLCToMotion.TechnologyObject.OutputCam.CathodeAlignVisionOutputCam := "Unit1.Em5.Config".outputCam[22];
END_REGION

REGION Network 308: Axis
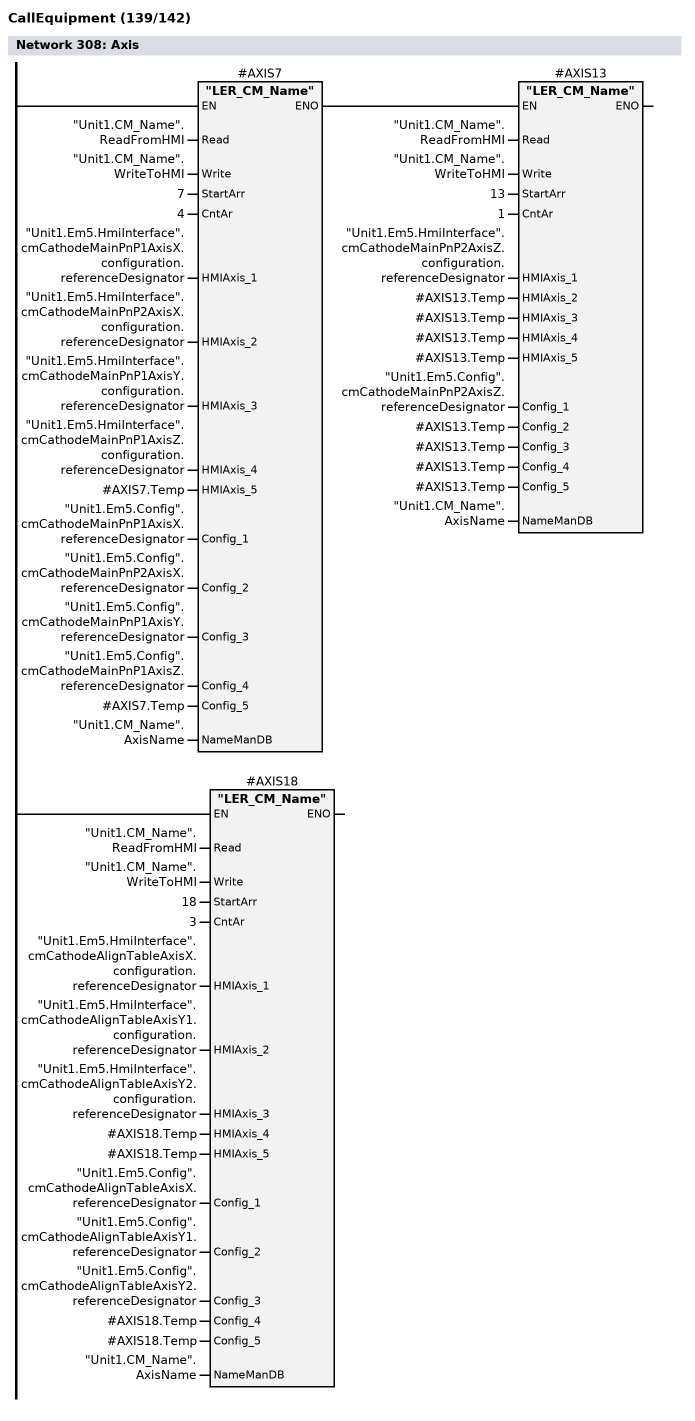
   RUNG wire#powerrail
      #AXIS7(Read := "Unit1.CM_Name".ReadFromHMI, Write := "Unit1.CM_Name".WriteToHMI, StartArr := 7, CntAr := 4, HMIAxis_1 := "Unit1.Em5.HmiInterface".cmCathodeMainPnP1AxisX.configuration.referenceDesignator, HMIAxis_2 := "Unit1.Em5.HmiInterface".cmCathodeMainPnP2AxisX.configuration.referenceDesignator, HMIAxis_3 := "Unit1.Em5.HmiInterface".cmCathodeMainPnP1AxisY.configuration.referenceDesignator, HMIAxis_4 := "Unit1.Em5.HmiInterface".cmCathodeMainPnP1AxisZ.configuration.referenceDesignator, HMIAxis_5 := #AXIS7.Temp, Config_1 := "Unit1.Em5.Config".cmCathodeMainPnP1AxisX.referenceDesignator, Config_2 := "Unit1.Em5.Config".cmCathodeMainPnP2AxisX.referenceDesignator, Config_3 := "Unit1.Em5.Config".cmCathodeMainPnP1AxisY.referenceDesignator, Config_4 := "Unit1.Em5.Config".cmCathodeMainPnP1AxisZ.referenceDesignator, Config_5 := #AXIS7.Temp, NameManDB := "Unit1.CM_Name".AxisName)
      #AXIS13(Read := "Unit1.CM_Name".ReadFromHMI, Write := "Unit1.CM_Name".WriteToHMI, StartArr := 13, CntAr := 1, HMIAxis_1 := "Unit1.Em5.HmiInterface".cmCathodeMainPnP2AxisZ.configuration.referenceDesignator, HMIAxis_2 := #AXIS13.Temp, HMIAxis_3 := #AXIS13.Temp, HMIAxis_4 := #AXIS13.Temp, HMIAxis_5 := #AXIS13.Temp, Config_1 := "Unit1.Em5.Config".cmCathodeMainPnP2AxisZ.referenceDesignator, Config_2 := #AXIS13.Temp, Config_3 := #AXIS13.Temp, Config_4 := #AXIS13.Temp, Config_5 := #AXIS13.Temp, NameManDB := "Unit1.CM_Name".AxisName)
   END_RUNG
   RUNG wire#powerrail
      #AXIS18(Read := "Unit1.CM_Name".ReadFromHMI, Write := "Unit1.CM_Name".WriteToHMI, StartArr := 18, CntAr := 3, HMIAxis_1 := "Unit1.Em5.HmiInterface".cmCathodeAlignTableAxisX.configuration.referenceDesignator, HMIAxis_2 := "Unit1.Em5.HmiInterface".cmCathodeAlignTableAxisY1.configuration.referenceDesignator, HMIAxis_3 := "Unit1.Em5.HmiInterface".cmCathodeAlignTableAxisY2.configuration.referenceDesignator, HMIAxis_4 := #AXIS18.Temp, HMIAxis_5 := #AXIS18.Temp, Config_1 := "Unit1.Em5.Config".cmCathodeAlignTableAxisX.referenceDesignator, Config_2 := "Unit1.Em5.Config".cmCathodeAlignTableAxisY1.referenceDesignator, Config_3 := "Unit1.Em5.Config".cmCathodeAlignTableAxisY2.referenceDesignator, Config_4 := #AXIS18.Temp, Config_5 := #AXIS18.Temp, NameManDB := "Unit1.CM_Name".AxisName)
   END_RUNG
   // the same network as SCL:
   #AXIS7(Read := "Unit1.CM_Name".ReadFromHMI,   // "LER_CM_Name"
          Write := "Unit1.CM_Name".WriteToHMI,
          StartArr := 7,
          CntAr := 4,
          HMIAxis_1 := "Unit1.Em5.HmiInterface".cmCathodeMainPnP1AxisX.configuration.referenceDesignator,
          HMIAxis_2 := "Unit1.Em5.HmiInterface".cmCathodeMainPnP2AxisX.configuration.referenceDesignator,
          HMIAxis_3 := "Unit1.Em5.HmiInterface".cmCathodeMainPnP1AxisY.configuration.referenceDesignator,
          HMIAxis_4 := "Unit1.Em5.HmiInterface".cmCathodeMainPnP1AxisZ.configuration.referenceDesignator,
          HMIAxis_5 := #AXIS7.Temp,
          Config_1 := "Unit1.Em5.Config".cmCathodeMainPnP1AxisX.referenceDesignator,
          Config_2 := "Unit1.Em5.Config".cmCathodeMainPnP2AxisX.referenceDesignator,
          Config_3 := "Unit1.Em5.Config".cmCathodeMainPnP1AxisY.referenceDesignator,
          Config_4 := "Unit1.Em5.Config".cmCathodeMainPnP1AxisZ.referenceDesignator,
          Config_5 := #AXIS7.Temp,
          NameManDB := "Unit1.CM_Name".AxisName,
          ENO => #_w1);
   IF #_w1 THEN
       #AXIS13(Read := "Unit1.CM_Name".ReadFromHMI,   // "LER_CM_Name"
               Write := "Unit1.CM_Name".WriteToHMI,
               StartArr := 13,
               CntAr := 1,
               HMIAxis_1 := "Unit1.Em5.HmiInterface".cmCathodeMainPnP2AxisZ.configuration.referenceDesignator,
               HMIAxis_2 := #AXIS13.Temp,
               HMIAxis_3 := #AXIS13.Temp,
               HMIAxis_4 := #AXIS13.Temp,
               HMIAxis_5 := #AXIS13.Temp,
               Config_1 := "Unit1.Em5.Config".cmCathodeMainPnP2AxisZ.referenceDesignator,
               Config_2 := #AXIS13.Temp,
               Config_3 := #AXIS13.Temp,
               Config_4 := #AXIS13.Temp,
               Config_5 := #AXIS13.Temp,
               NameManDB := "Unit1.CM_Name".AxisName);
   END_IF;
   #AXIS18(Read := "Unit1.CM_Name".ReadFromHMI,   // "LER_CM_Name"
           Write := "Unit1.CM_Name".WriteToHMI,
           StartArr := 18,
           CntAr := 3,
           HMIAxis_1 := "Unit1.Em5.HmiInterface".cmCathodeAlignTableAxisX.configuration.referenceDesignator,
           HMIAxis_2 := "Unit1.Em5.HmiInterface".cmCathodeAlignTableAxisY1.configuration.referenceDesignator,
           HMIAxis_3 := "Unit1.Em5.HmiInterface".cmCathodeAlignTableAxisY2.configuration.referenceDesignator,
           HMIAxis_4 := #AXIS18.Temp,
           HMIAxis_5 := #AXIS18.Temp,
           Config_1 := "Unit1.Em5.Config".cmCathodeAlignTableAxisX.referenceDesignator,
           Config_2 := "Unit1.Em5.Config".cmCathodeAlignTableAxisY1.referenceDesignator,
           Config_3 := "Unit1.Em5.Config".cmCathodeAlignTableAxisY2.referenceDesignator,
           Config_4 := #AXIS18.Temp,
           Config_5 := #AXIS18.Temp,
           NameManDB := "Unit1.CM_Name".AxisName);
END_REGION

REGION Network 309: Cylinder
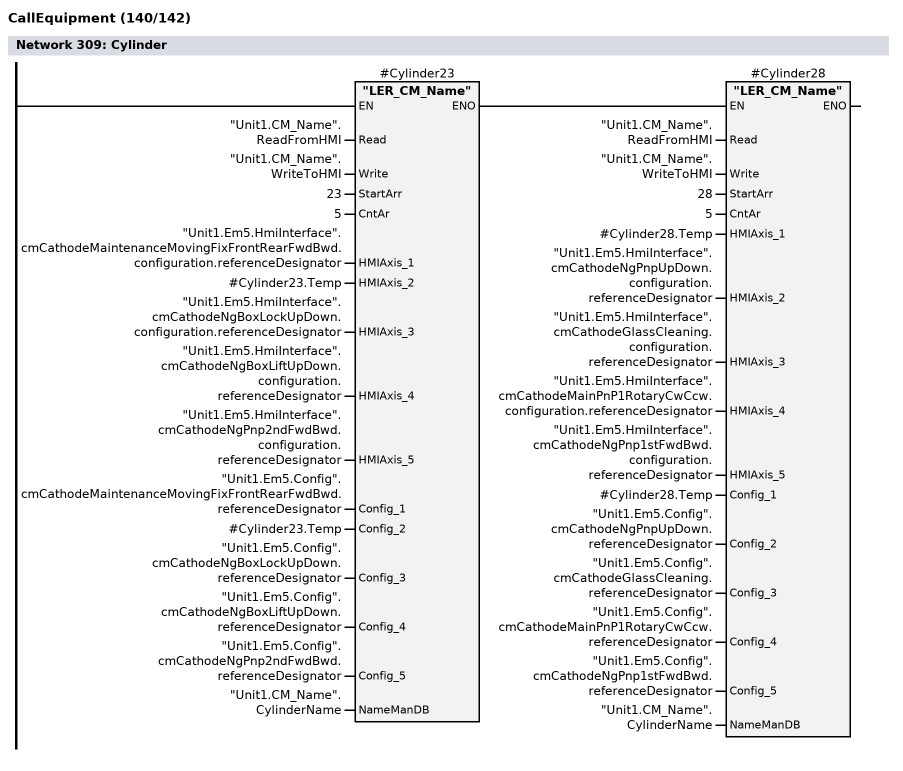
   RUNG wire#powerrail
      #Cylinder23(Read := "Unit1.CM_Name".ReadFromHMI, Write := "Unit1.CM_Name".WriteToHMI, StartArr := 23, CntAr := 5, HMIAxis_1 := "Unit1.Em5.HmiInterface".cmCathodeMaintenanceMovingFixFrontRearFwdBwd.configuration.referenceDesignator, HMIAxis_2 := #Cylinder23.Temp, HMIAxis_3 := "Unit1.Em5.HmiInterface".cmCathodeNgBoxLockUpDown.configuration.referenceDesignator, HMIAxis_4 := "Unit1.Em5.HmiInterface".cmCathodeNgBoxLiftUpDown.configuration.referenceDesignator, HMIAxis_5 := "Unit1.Em5.HmiInterface".cmCathodeNgPnp2ndFwdBwd.configuration.referenceDesignator, Config_1 := "Unit1.Em5.Config".cmCathodeMaintenanceMovingFixFrontRearFwdBwd.referenceDesignator, Config_2 := #Cylinder23.Temp, Config_3 := "Unit1.Em5.Config".cmCathodeNgBoxLockUpDown.referenceDesignator, Config_4 := "Unit1.Em5.Config".cmCathodeNgBoxLiftUpDown.referenceDesignator, Config_5 := "Unit1.Em5.Config".cmCathodeNgPnp2ndFwdBwd.referenceDesignator, NameManDB := "Unit1.CM_Name".CylinderName)
      #Cylinder28(Read := "Unit1.CM_Name".ReadFromHMI, Write := "Unit1.CM_Name".WriteToHMI, StartArr := 28, CntAr := 5, HMIAxis_1 := #Cylinder28.Temp, HMIAxis_2 := "Unit1.Em5.HmiInterface".cmCathodeNgPnpUpDown.configuration.referenceDesignator, HMIAxis_3 := "Unit1.Em5.HmiInterface".cmCathodeGlassCleaning.configuration.referenceDesignator, HMIAxis_4 := "Unit1.Em5.HmiInterface".cmCathodeMainPnP1RotaryCwCcw.configuration.referenceDesignator, HMIAxis_5 := "Unit1.Em5.HmiInterface".cmCathodeNgPnp1stFwdBwd.configuration.referenceDesignator, Config_1 := #Cylinder28.Temp, Config_2 := "Unit1.Em5.Config".cmCathodeNgPnpUpDown.referenceDesignator, Config_3 := "Unit1.Em5.Config".cmCathodeGlassCleaning.referenceDesignator, Config_4 := "Unit1.Em5.Config".cmCathodeMainPnP1RotaryCwCcw.referenceDesignator, Config_5 := "Unit1.Em5.Config".cmCathodeNgPnp1stFwdBwd.referenceDesignator, NameManDB := "Unit1.CM_Name".CylinderName)
   END_RUNG
   // the same network as SCL:
   #Cylinder23(Read := "Unit1.CM_Name".ReadFromHMI,   // "LER_CM_Name"
               Write := "Unit1.CM_Name".WriteToHMI,
               StartArr := 23,
               CntAr := 5,
               HMIAxis_1 := "Unit1.Em5.HmiInterface".cmCathodeMaintenanceMovingFixFrontRearFwdBwd.configuration.referenceDesignator,
               HMIAxis_2 := #Cylinder23.Temp,
               HMIAxis_3 := "Unit1.Em5.HmiInterface".cmCathodeNgBoxLockUpDown.configuration.referenceDesignator,
               HMIAxis_4 := "Unit1.Em5.HmiInterface".cmCathodeNgBoxLiftUpDown.configuration.referenceDesignator,
               HMIAxis_5 := "Unit1.Em5.HmiInterface".cmCathodeNgPnp2ndFwdBwd.configuration.referenceDesignator,
               Config_1 := "Unit1.Em5.Config".cmCathodeMaintenanceMovingFixFrontRearFwdBwd.referenceDesignator,
               Config_2 := #Cylinder23.Temp,
               Config_3 := "Unit1.Em5.Config".cmCathodeNgBoxLockUpDown.referenceDesignator,
               Config_4 := "Unit1.Em5.Config".cmCathodeNgBoxLiftUpDown.referenceDesignator,
               Config_5 := "Unit1.Em5.Config".cmCathodeNgPnp2ndFwdBwd.referenceDesignator,
               NameManDB := "Unit1.CM_Name".CylinderName,
               ENO => #_w1);
   IF #_w1 THEN
       #Cylinder28(Read := "Unit1.CM_Name".ReadFromHMI,   // "LER_CM_Name"
                   Write := "Unit1.CM_Name".WriteToHMI,
                   StartArr := 28,
                   CntAr := 5,
                   HMIAxis_1 := #Cylinder28.Temp,
                   HMIAxis_2 := "Unit1.Em5.HmiInterface".cmCathodeNgPnpUpDown.configuration.referenceDesignator,
                   HMIAxis_3 := "Unit1.Em5.HmiInterface".cmCathodeGlassCleaning.configuration.referenceDesignator,
                   HMIAxis_4 := "Unit1.Em5.HmiInterface".cmCathodeMainPnP1RotaryCwCcw.configuration.referenceDesignator,
                   HMIAxis_5 := "Unit1.Em5.HmiInterface".cmCathodeNgPnp1stFwdBwd.configuration.referenceDesignator,
                   Config_1 := #Cylinder28.Temp,
                   Config_2 := "Unit1.Em5.Config".cmCathodeNgPnpUpDown.referenceDesignator,
                   Config_3 := "Unit1.Em5.Config".cmCathodeGlassCleaning.referenceDesignator,
                   Config_4 := "Unit1.Em5.Config".cmCathodeMainPnP1RotaryCwCcw.referenceDesignator,
                   Config_5 := "Unit1.Em5.Config".cmCathodeNgPnp1stFwdBwd.referenceDesignator,
                   NameManDB := "Unit1.CM_Name".CylinderName);
   END_IF;
END_REGION

REGION Network 310: Vaccum
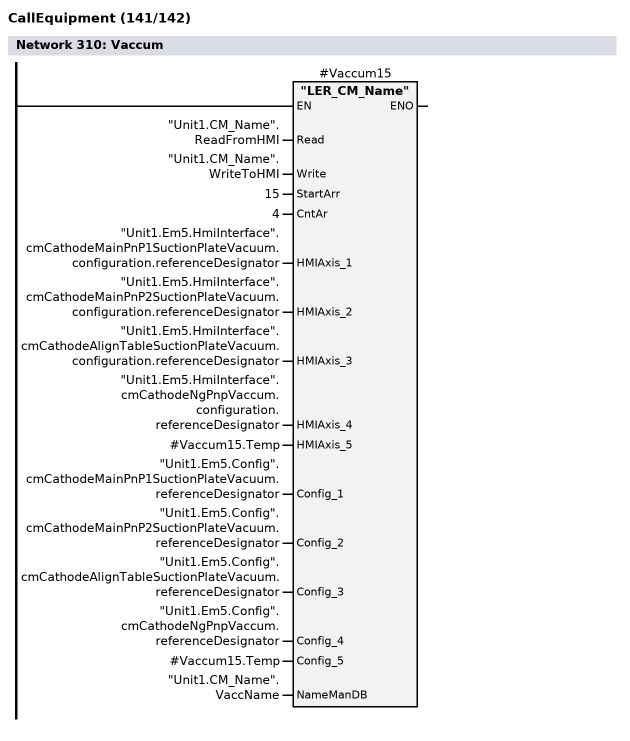
   RUNG wire#powerrail
      #Vaccum15(Read := "Unit1.CM_Name".ReadFromHMI, Write := "Unit1.CM_Name".WriteToHMI, StartArr := 15, CntAr := 4, HMIAxis_1 := "Unit1.Em5.HmiInterface".cmCathodeMainPnP1SuctionPlateVacuum.configuration.referenceDesignator, HMIAxis_2 := "Unit1.Em5.HmiInterface".cmCathodeMainPnP2SuctionPlateVacuum.configuration.referenceDesignator, HMIAxis_3 := "Unit1.Em5.HmiInterface".cmCathodeAlignTableSuctionPlateVacuum.configuration.referenceDesignator, HMIAxis_4 := "Unit1.Em5.HmiInterface".cmCathodeNgPnpVaccum.configuration.referenceDesignator, HMIAxis_5 := #Vaccum15.Temp, Config_1 := "Unit1.Em5.Config".cmCathodeMainPnP1SuctionPlateVacuum.referenceDesignator, Config_2 := "Unit1.Em5.Config".cmCathodeMainPnP2SuctionPlateVacuum.referenceDesignator, Config_3 := "Unit1.Em5.Config".cmCathodeAlignTableSuctionPlateVacuum.referenceDesignator, Config_4 := "Unit1.Em5.Config".cmCathodeNgPnpVaccum.referenceDesignator, Config_5 := #Vaccum15.Temp, NameManDB := "Unit1.CM_Name".VaccName)
   END_RUNG
   // the same network as SCL:
   #Vaccum15(Read := "Unit1.CM_Name".ReadFromHMI,   // "LER_CM_Name"
             Write := "Unit1.CM_Name".WriteToHMI,
             StartArr := 15,
             CntAr := 4,
             HMIAxis_1 := "Unit1.Em5.HmiInterface".cmCathodeMainPnP1SuctionPlateVacuum.configuration.referenceDesignator,
             HMIAxis_2 := "Unit1.Em5.HmiInterface".cmCathodeMainPnP2SuctionPlateVacuum.configuration.referenceDesignator,
             HMIAxis_3 := "Unit1.Em5.HmiInterface".cmCathodeAlignTableSuctionPlateVacuum.configuration.referenceDesignator,
             HMIAxis_4 := "Unit1.Em5.HmiInterface".cmCathodeNgPnpVaccum.configuration.referenceDesignator,
             HMIAxis_5 := #Vaccum15.Temp,
             Config_1 := "Unit1.Em5.Config".cmCathodeMainPnP1SuctionPlateVacuum.referenceDesignator,
             Config_2 := "Unit1.Em5.Config".cmCathodeMainPnP2SuctionPlateVacuum.referenceDesignator,
             Config_3 := "Unit1.Em5.Config".cmCathodeAlignTableSuctionPlateVacuum.referenceDesignator,
             Config_4 := "Unit1.Em5.Config".cmCathodeNgPnpVaccum.referenceDesignator,
             Config_5 := #Vaccum15.Temp,
             NameManDB := "Unit1.CM_Name".VaccName);
END_REGION

REGION Network 311: BA010 Interface Data
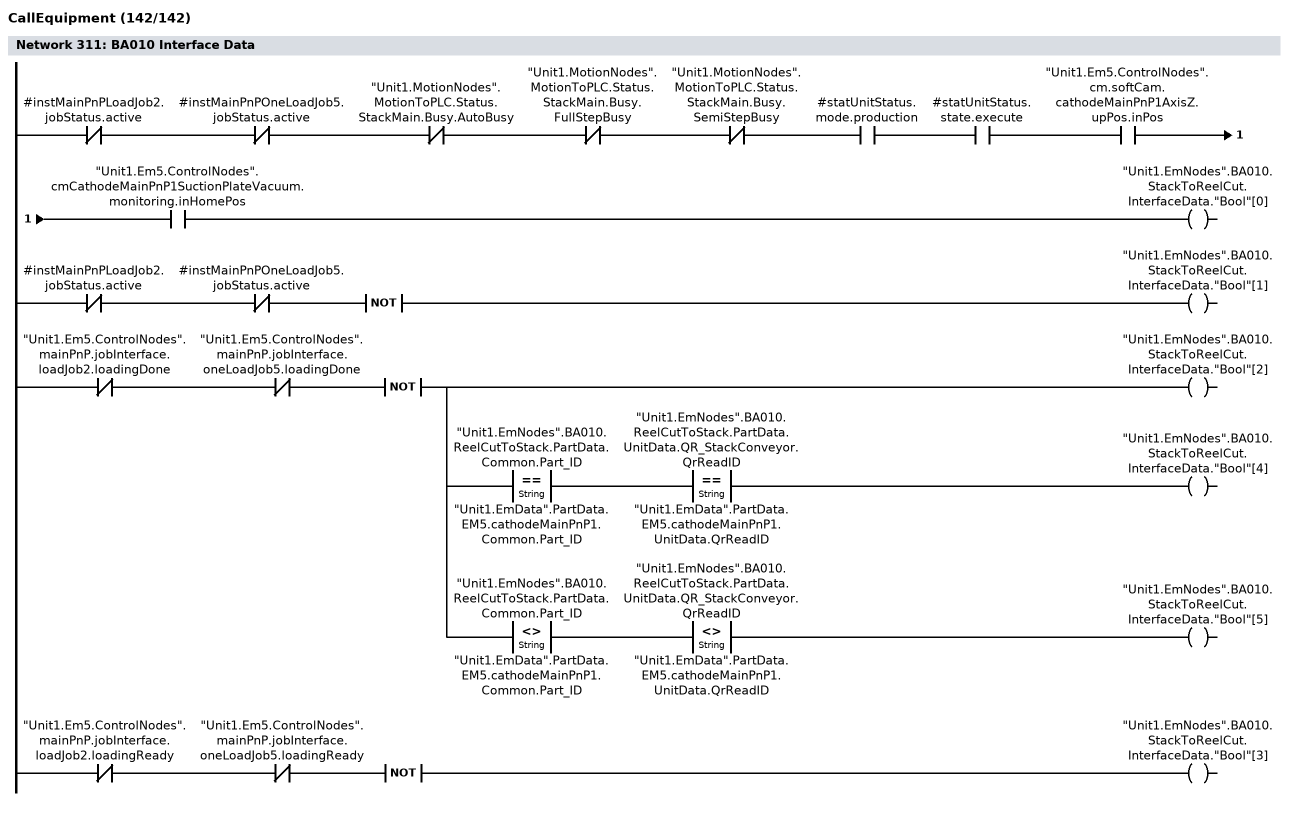
   RUNG wire#powerrail
      I_Contact( #instMainPnPLoadJob2.jobStatus.active )
      I_Contact( #instMainPnPOneLoadJob5.jobStatus.active )
      I_Contact( "Unit1.MotionNodes".MotionToPLC.Status.StackMain.Busy.AutoBusy )
      I_Contact( "Unit1.MotionNodes".MotionToPLC.Status.StackMain.Busy.FullStepBusy )
      I_Contact( "Unit1.MotionNodes".MotionToPLC.Status.StackMain.Busy.SemiStepBusy )
      Contact( #statUnitStatus.mode.production )
      Contact( #statUnitStatus.state.execute )
      Contact( "Unit1.Em5.ControlNodes".cm.softCam.cathodeMainPnP1AxisZ.upPos.inPos )
      Contact( "Unit1.Em5.ControlNodes".cmCathodeMainPnP1SuctionPlateVacuum.monitoring.inHomePos )
      Coil( "Unit1.EmNodes".BA010.StackToReelCut.InterfaceData."Bool"[0] )
   END_RUNG
   RUNG wire#powerrail
      I_Contact( #instMainPnPLoadJob2.jobStatus.active )
      I_Contact( #instMainPnPOneLoadJob5.jobStatus.active )
      Not()
      Coil( "Unit1.EmNodes".BA010.StackToReelCut.InterfaceData."Bool"[1] )
   END_RUNG
   RUNG wire#powerrail
      I_Contact( "Unit1.Em5.ControlNodes".mainPnP.jobInterface.loadJob2.loadingDone )
      I_Contact( "Unit1.Em5.ControlNodes".mainPnP.jobInterface.oneLoadJob5.loadingDone )
      Not()
      wire#w1
      Coil( "Unit1.EmNodes".BA010.StackToReelCut.InterfaceData."Bool"[2] )
   END_RUNG
   RUNG wire#w1
      { S7_Templates := "SrcType := String" } EQ_Contact(in1 := "Unit1.EmNodes".BA010.ReelCutToStack.PartData.Common.Part_ID, in2 := "Unit1.EmData".PartData.EM5.cathodeMainPnP1.Common.Part_ID)
      { S7_Templates := "SrcType := String" } EQ_Contact(in1 := "Unit1.EmNodes".BA010.ReelCutToStack.PartData.UnitData.QR_StackConveyor.QrReadID, in2 := "Unit1.EmData".PartData.EM5.cathodeMainPnP1.UnitData.QrReadID)
      Coil( "Unit1.EmNodes".BA010.StackToReelCut.InterfaceData."Bool"[4] )
   END_RUNG
   RUNG wire#w1
      { S7_Templates := "SrcType := String" } NE_Contact(in1 := "Unit1.EmNodes".BA010.ReelCutToStack.PartData.Common.Part_ID, in2 := "Unit1.EmData".PartData.EM5.cathodeMainPnP1.Common.Part_ID)
      { S7_Templates := "SrcType := String" } NE_Contact(in1 := "Unit1.EmNodes".BA010.ReelCutToStack.PartData.UnitData.QR_StackConveyor.QrReadID, in2 := "Unit1.EmData".PartData.EM5.cathodeMainPnP1.UnitData.QrReadID)
      Coil( "Unit1.EmNodes".BA010.StackToReelCut.InterfaceData."Bool"[5] )
   END_RUNG
   RUNG wire#powerrail
      I_Contact( "Unit1.Em5.ControlNodes".mainPnP.jobInterface.loadJob2.loadingReady )
      I_Contact( "Unit1.Em5.ControlNodes".mainPnP.jobInterface.oneLoadJob5.loadingReady )
      Not()
      Coil( "Unit1.EmNodes".BA010.StackToReelCut.InterfaceData."Bool"[3] )
   END_RUNG
   // the same network as SCL:
   "Unit1.EmNodes".BA010.StackToReelCut.InterfaceData."Bool"[0] := NOT #instMainPnPLoadJob2.jobStatus.active AND NOT #instMainPnPOneLoadJob5.jobStatus.active AND NOT "Unit1.MotionNodes".MotionToPLC.Status.StackMain.Busy.AutoBusy AND NOT "Unit1.MotionNodes".MotionToPLC.Status.StackMain.Busy.FullStepBusy AND NOT "Unit1.MotionNodes".MotionToPLC.Status.StackMain.Busy.SemiStepBusy AND #statUnitStatus.mode.production AND #statUnitStatus.state.execute AND "Unit1.Em5.ControlNodes".cm.softCam.cathodeMainPnP1AxisZ.upPos.inPos AND "Unit1.Em5.ControlNodes".cmCathodeMainPnP1SuctionPlateVacuum.monitoring.inHomePos;
   "Unit1.EmNodes".BA010.StackToReelCut.InterfaceData."Bool"[1] := NOT (NOT #instMainPnPLoadJob2.jobStatus.active AND NOT #instMainPnPOneLoadJob5.jobStatus.active);
   "Unit1.EmNodes".BA010.StackToReelCut.InterfaceData."Bool"[2] := NOT (NOT "Unit1.Em5.ControlNodes".mainPnP.jobInterface.loadJob2.loadingDone AND NOT "Unit1.Em5.ControlNodes".mainPnP.jobInterface.oneLoadJob5.loadingDone);
   "Unit1.EmNodes".BA010.StackToReelCut.InterfaceData."Bool"[4] := NOT (NOT "Unit1.Em5.ControlNodes".mainPnP.jobInterface.loadJob2.loadingDone AND NOT "Unit1.Em5.ControlNodes".mainPnP.jobInterface.oneLoadJob5.loadingDone) AND ("Unit1.EmNodes".BA010.ReelCutToStack.PartData.Common.Part_ID = "Unit1.EmData".PartData.EM5.cathodeMainPnP1.Common.Part_ID) AND ("Unit1.EmNodes".BA010.ReelCutToStack.PartData.UnitData.QR_StackConveyor.QrReadID = "Unit1.EmData".PartData.EM5.cathodeMainPnP1.UnitData.QrReadID);
   "Unit1.EmNodes".BA010.StackToReelCut.InterfaceData."Bool"[5] := NOT (NOT "Unit1.Em5.ControlNodes".mainPnP.jobInterface.loadJob2.loadingDone AND NOT "Unit1.Em5.ControlNodes".mainPnP.jobInterface.oneLoadJob5.loadingDone) AND ("Unit1.EmNodes".BA010.ReelCutToStack.PartData.Common.Part_ID <> "Unit1.EmData".PartData.EM5.cathodeMainPnP1.Common.Part_ID) AND ("Unit1.EmNodes".BA010.ReelCutToStack.PartData.UnitData.QR_StackConveyor.QrReadID <> "Unit1.EmData".PartData.EM5.cathodeMainPnP1.UnitData.QrReadID);
   "Unit1.EmNodes".BA010.StackToReelCut.InterfaceData."Bool"[3] := NOT (NOT "Unit1.Em5.ControlNodes".mainPnP.jobInterface.loadJob2.loadingReady AND NOT "Unit1.Em5.ControlNodes".mainPnP.jobInterface.oneLoadJob5.loadingReady);
END_REGION
END_FUNCTION_BLOCK
